KUKA KRL program: MyProgram_229().src

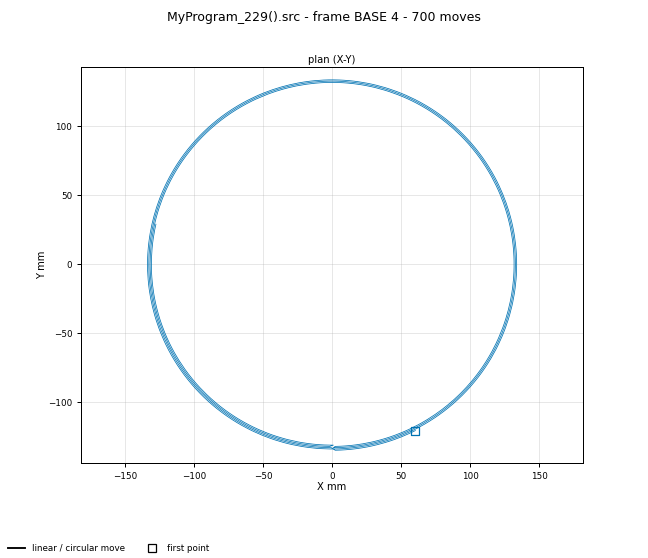
[picture p0: tool path of MyProgram_229().src in frame BASE 4, 700 of 700 moves have a stored position in this frame; points joined in program order, loops and branches not executed]
&ACCESS RVP
&REL 1
&PARAM TEMPLATE = C:\KRC\Roboter\Template\vorgabe
&PARAM EDITMASK = *
DEF MyProgram_229()
; ---- Setting reference (Base) ----
$BASE = BASE_DATA[4]

; --------------------------
; ---- Setting tool (TCP) ----
$TOOL = TOOL_DATA[3]
; --------------------------

$VEL.CP = VEL_APROX_PRINT
Startdeposition()
$VEL.CP = VEL_PRINT
LIN {X 60.3431,Y -120.4102,Z 157,A -66.3783,B 23.115,C -0.9424,E1 23.2036,E2 513.6241} C_DIS
LIN {X 55.6894,Y -122.6317,Z 157,A -68.3242,B 23.1147,C -0.9514,E1 23.1988,E2 515.5416} C_DIS
LIN {X 53.1438,Y -123.7542,Z 157,A -69.519,B 23.1147,C -0.9491,E1 23.1957,E2 516.7391} C_DIS
LIN {X 50.0848,Y -125.0234,Z 157,A -70.9751,B 23.1149,C -0.9447,E1 23.1919,E2 518.2027} C_DIS
LIN {X 44.88,Y -126.987,Z 157,A -73.2835,B 23.1149,C -0.9444,E1 23.1859,E2 520.5065} C_DIS
LIN {X 42.2863,Y -127.8719,Z 157,A -74.8329,B 23.1157,C -0.9239,E1 23.1816,E2 522.1048} C_DIS
LIN {X 38.6503,Y -129.0197,Z 157,A -76.0668,B 23.1151,C -0.9413,E1 23.1785,E2 523.292} C_DIS
LIN {X 32.9154,Y -130.5983,Z 157,A -78.6147,B 23.1151,C -0.9378,E1 23.1716,E2 525.8445} C_DIS
LIN {X 29.0818,Y -131.5067,Z 157,A -80.3833,B 23.1154,C -0.9316,E1 23.1667,E2 527.6262} C_DIS
LIN {X 25.3199,Y -132.2809,Z 157,A -81.9079,B 23.1153,C -0.9357,E1 23.1626,E2 529.1385} C_DIS
LIN {X 21.8715,Y -132.8949,Z 157,A -83.4811,B 23.1155,C -0.9304,E1 23.1582,E2 530.7233} C_DIS
LIN {X 17.6299,Y -133.5236,Z 157,A -85.227,B 23.1154,C -0.933,E1 23.1534,E2 532.4607} C_DIS
LIN {X 14.202,Y -133.9317,Z 157,A -86.7009,B 23.1154,C -0.9319,E1 23.1493,E2 533.9363} C_DIS
LIN {X 10.0398,Y -134.308,Z 157,A -88.4861,B 23.1154,C -0.9307,E1 23.1444,E2 535.7236} C_DIS
LIN {X 6.4164,Y -134.53,Z 157,A -90.0918,B 23.1156,C -0.9271,E1 23.1399,E2 537.3379} C_DIS
LIN {X 2.2217,Y -134.6642,Z 157,A -91.783,B 23.1154,C -0.9312,E1 23.1352,E2 539.0183} C_DIS
LIN {X 2.2217,Y -134.6642,Z 157,A -91.783,B 23.1154,C -0.9312,E1 23.1352,E2 539.0183} C_DIS
Enddeposition()
LIN {X 0.9379,Y -133.7479,Z 157,A -91.7114,B 21.9007,C -0.7569,E1 21.9144,E2 539.2658} C_DIS
Startdeposition()
$VEL.CP = VEL_PRINT
LIN {X 5.092,Y -133.6541,Z 157,A -89.5299,B 21.9,C -0.776,E1 21.9206,E2 537.0334} C_DIS
LIN {X 8.4927,Y -133.4814,Z 157,A -88.065,B 21.9,C -0.7769,E1 21.9247,E2 535.5668} C_DIS
LIN {X 12.2431,Y -133.1905,Z 157,A -86.4619,B 21.9,C -0.7773,E1 21.9292,E2 533.9638} C_DIS
LIN {X 15.7185,Y -132.8241,Z 157,A -84.992,B 21.9,C -0.7769,E1 21.9333,E2 532.4962} C_DIS
LIN {X 18.8317,Y -132.4185,Z 157,A -83.651,B 21.9,C -0.7775,E1 21.937,E2 531.1547} C_DIS
LIN {X 22.9546,Y -131.7678,Z 157,A -81.9321,B 21.9,C -0.7756,E1 21.9417,E2 529.4432} C_DIS
LIN {X 25.8918,Y -131.2232,Z 157,A -80.5104,B 21.8998,C -0.7833,E1 21.9456,E2 528.0027} C_DIS
LIN {X 29.3532,Y -130.4908,Z 157,A -79.0266,B 21.8998,C -0.7832,E1 21.9497,E2 526.5215} C_DIS
LIN {X 32.3293,Y -129.786,Z 157,A -77.8447,B 21.9,C -0.7783,E1 21.9528,E2 525.3545} C_DIS
LIN {X 35.2431,Y -129.0264,Z 157,A -76.4748,B 21.8998,C -0.7834,E1 21.9566,E2 523.9735} C_DIS
LIN {X 38.3629,Y -128.1335,Z 157,A -75.0868,B 21.8998,C -0.7849,E1 21.9603,E2 522.5844} C_DIS
LIN {X 41.4791,Y -127.1589,Z 157,A -73.6902,B 21.8997,C -0.7864,E1 21.964,E2 521.1866} C_DIS
LIN {X 45.073,Y -125.9275,Z 157,A -72.1814,B 21.8998,C -0.7828,E1 21.968,E2 519.691} C_DIS
LIN {X 47.6885,Y -124.9628,Z 157,A -70.8737,B 21.8996,C -0.7898,E1 21.9714,E2 518.3679} C_DIS
LIN {X 51.0833,Y -123.6121,Z 157,A -69.2486,B 21.8994,C -0.7949,E1 21.9756,E2 516.7335} C_DIS
LIN {X 54.2918,Y -122.2364,Z 157,A -68.0057,B 21.8997,C -0.785,E1 21.9787,E2 515.5205} C_DIS
LIN {X 56.898,Y -121.0476,Z 157,A -66.5962,B 21.8994,C -0.7956,E1 21.9824,E2 514.0869} C_DIS
LIN {X 59.9271,Y -119.577,Z 157,A -65.158,B 21.8994,C -0.7977,E1 21.986,E2 512.6475} C_DIS
LIN {X 63.2603,Y -117.8468,Z 157,A -63.4648,B 21.8991,C -0.8045,E1 21.9902,E2 510.9417} C_DIS
LIN {X 66.9687,Y -115.7796,Z 157,A -61.6672,B 21.899,C -0.8067,E1 21.9946,E2 509.1444} C_DIS
LIN {X 70.6246,Y -113.5865,Z 157,A -59.8473,B 21.8989,C -0.8097,E1 21.9989,E2 507.323} C_DIS
LIN {X 74.4235,Y -111.1346,Z 157,A -57.9624,B 21.8989,C -0.811,E1 22.0033,E2 505.442} C_DIS
LIN {X 77.7542,Y -108.8301,Z 157,A -56.1901,B 21.8987,C -0.8163,E1 22.0073,E2 503.6626} C_DIS
LIN {X 81.2948,Y -106.2115,Z 157,A -54.3316,B 21.8986,C -0.8189,E1 22.0115,E2 501.805} C_DIS
LIN {X 84.6122,Y -103.588,Z 157,A -52.512,B 21.8984,C -0.8232,E1 22.0155,E2 499.9819} C_DIS
LIN {X 87.977,Y -100.746,Z 157,A -50.6512,B 21.8983,C -0.8262,E1 22.0194,E2 498.1215} C_DIS
LIN {X 91.1152,Y -97.917,Z 157,A -48.8313,B 21.8981,C -0.8308,E1 22.0232,E2 496.2977} C_DIS
LIN {X 94.3364,Y -94.8176,Z 157,A -46.9545,B 21.8981,C -0.8336,E1 22.0269,E2 494.4228} C_DIS
LIN {X 97.2567,Y -91.8196,Z 157,A -45.1448,B 21.8978,C -0.8388,E1 22.0304,E2 492.6081} C_DIS
LIN {X 100.1751,Y -88.6266,Z 157,A -43.303,B 21.8977,C -0.8429,E1 22.0338,E2 490.7649} C_DIS
LIN {X 103.0497,Y -85.2671,Z 157,A -41.4192,B 21.8975,C -0.8473,E1 22.0372,E2 488.8793} C_DIS
LIN {X 105.6853,Y -81.9776,Z 157,A -39.6275,B 21.8974,C -0.8514,E1 22.0403,E2 487.0864} C_DIS
LIN {X 108.3279,Y -78.4524,Z 157,A -37.7727,B 21.8972,C -0.8549,E1 22.0434,E2 485.2326} C_DIS
LIN {X 110.867,Y -74.8216,Z 157,A -35.9119,B 21.8972,C -0.8583,E1 22.0464,E2 483.3734} C_DIS
LIN {X 113.1329,Y -71.349,Z 157,A -34.1251,B 21.8969,C -0.8638,E1 22.0491,E2 481.5822} C_DIS
LIN {X 115.3011,Y -67.7892,Z 157,A -32.3337,B 21.8967,C -0.8692,E1 22.0516,E2 479.7871} C_DIS
LIN {X 117.4775,Y -63.9435,Z 157,A -30.5231,B 21.8967,C -0.8706,E1 22.0541,E2 477.9836} C_DIS
LIN {X 118.8108,Y -61.4321,Z 157,A -29.1905,B 21.8963,C -0.8799,E1 22.0558,E2 476.6346} C_DIS
LIN {X 120.4363,Y -58.1775,Z 157,A -27.7272,B 21.8963,C -0.8799,E1 22.0576,E2 475.1805} C_DIS
LIN {X 121.9368,Y -54.9615,Z 157,A -26.4378,B 21.8966,C -0.873,E1 22.0591,E2 473.9175} C_DIS
LIN {X 123.0985,Y -52.3132,Z 157,A -25.038,B 21.8961,C -0.8847,E1 22.0606,E2 472.4954} C_DIS
LIN {X 124.3621,Y -49.2338,Z 157,A -23.6241,B 21.896,C -0.8884,E1 22.0621,E2 471.0806} C_DIS
LIN {X 125.5428,Y -46.14,Z 157,A -22.1041,B 21.8956,C -0.8978,E1 22.0636,E2 469.5453} C_DIS
LIN {X 126.7948,Y -42.5725,Z 157,A -20.796,B 21.896,C -0.8874,E1 22.0648,E2 468.2734} C_DIS
LIN {X 127.6564,Y -39.9216,Z 157,A -19.4281,B 21.8955,C -0.8997,E1 22.066,E2 466.8818} C_DIS
LIN {X 128.6609,Y -36.5501,Z 157,A -17.8608,B 21.8952,C -0.9075,E1 22.0672,E2 465.3042} C_DIS
LIN {X 129.5424,Y -33.2894,Z 157,A -16.4631,B 21.8952,C -0.9096,E1 22.0682,E2 463.9101} C_DIS
LIN {X 130.3092,Y -30.1481,Z 157,A -15.1727,B 21.8952,C -0.9093,E1 22.069,E2 462.6291} C_DIS
LIN {X 130.9066,Y -27.4474,Z 157,A -13.9534,B 21.8949,C -0.9147,E1 22.0697,E2 461.4036} C_DIS
LIN {X 131.6022,Y -23.8795,Z 157,A -12.5864,B 21.8951,C -0.9103,E1 22.0704,E2 460.0576} C_DIS
LIN {X 132.0562,Y -21.238,Z 157,A -11.2094,B 21.8945,C -0.9253,E1 22.0711,E2 458.6501} C_DIS
LIN {X 132.5855,Y -17.6196,Z 157,A -9.7043,B 21.8945,C -0.9273,E1 22.0716,E2 457.1499} C_DIS
LIN {X 132.9737,Y -14.3987,Z 157,A -8.3451,B 21.8943,C -0.9303,E1 22.0721,E2 455.7922} C_DIS
LIN {X 133.2838,Y -11.1695,Z 157,A -6.9683,B 21.8942,C -0.9341,E1 22.0724,E2 454.4146} C_DIS
LIN {X 133.5189,Y -7.8835,Z 157,A -5.4562,B 21.8938,C -0.9436,E1 22.0727,E2 452.8876} C_DIS
LIN {X 133.697,Y -3.8022,Z 157,A -3.7923,B 21.8938,C -0.945,E1 22.0729,E2 451.2314} C_DIS
LIN {X 133.7532,Y -0.2268,Z 157,A -2.1342,B 21.8933,C -0.9561,E1 22.0729,E2 449.5551} C_DIS
LIN {X 133.7072,Y 3.4346,Z 157,A -0.713,B 21.8933,C -0.9539,E1 22.0729,E2 448.1497} C_DIS
LIN {X 133.5779,Y 6.8027,Z 157,A 0.707,B 21.8933,C -0.9573,E1 22.0726,E2 446.7303} C_DIS
LIN {X 133.3249,Y 10.683,Z 157,A 2.434,B 21.8929,C -0.9657,E1 22.0723,E2 444.993} C_DIS
LIN {X 132.9986,Y 14.1666,Z 157,A 3.8365,B 21.8929,C -0.9657,E1 22.0719,E2 443.6} C_DIS
LIN {X 132.6097,Y 17.4345,Z 157,A 5.1979,B 21.8928,C -0.9678,E1 22.0714,E2 442.2424} C_DIS
LIN {X 132.1802,Y 20.4373,Z 157,A 6.5397,B 21.8925,C -0.9739,E1 22.0709,E2 440.8933} C_DIS
LIN {X 131.6149,Y 23.8088,Z 157,A 8.0257,B 21.8923,C -0.9796,E1 22.0702,E2 439.4023} C_DIS
LIN {X 130.9066,Y 27.4474,Z 157,A 9.5524,B 21.8923,C -0.9815,E1 22.0693,E2 437.881} C_DIS
LIN {X 130.2144,Y 30.5633,Z 157,A 11.0415,B 21.8918,C -0.9917,E1 22.0684,E2 436.3745} C_DIS
LIN {X 129.301,Y 34.2137,Z 157,A 12.5379,B 21.8918,C -0.991,E1 22.0673,E2 434.8902} C_DIS
LIN {X 128.1335,Y 38.3629,Z 157,A 14.3501,B 21.8916,C -0.9949,E1 22.0659,E2 433.0796} C_DIS
LIN {X 127.0837,Y 41.7048,Z 157,A 15.7518,B 21.8916,C -0.9945,E1 22.0647,E2 431.688} C_DIS
LIN {X 126.1021,Y 44.5887,Z 157,A 17.2854,B 21.891,C -1.0096,E1 22.0633,E2 430.1242} C_DIS
LIN {X 124.7807,Y 48.1571,Z 157,A 18.7673,B 21.891,C -1.0072,E1 22.0619,E2 428.6583} C_DIS
LIN {X 123.607,Y 51.0956,Z 157,A 20.1147,B 21.891,C -1.0107,E1 22.0604,E2 427.3102} C_DIS
LIN {X 122.3341,Y 54.0731,Z 157,A 21.4435,B 21.8909,C -1.0118,E1 22.059,E2 425.9867} C_DIS
LIN {X 121.0476,Y 56.898,Z 157,A 22.8092,B 21.8906,C -1.0173,E1 22.0573,E2 424.615} C_DIS
LIN {X 119.577,Y 59.9271,Z 157,A 24.2433,B 21.8905,C -1.021,E1 22.0556,E2 423.1801} C_DIS
LIN {X 117.8468,Y 63.2603,Z 157,A 25.9173,B 21.8901,C -1.0286,E1 22.0534,E2 421.496} C_DIS
LIN {X 115.7796,Y 66.9687,Z 157,A 27.7258,B 21.8899,C -1.033,E1 22.0509,E2 419.6865} C_DIS
LIN {X 113.5117,Y 70.7447,Z 157,A 29.5907,B 21.8898,C -1.0369,E1 22.0482,E2 417.8221} C_DIS
LIN {X 111.2141,Y 74.3044,Z 157,A 31.3882,B 21.8896,C -1.0408,E1 22.0454,E2 416.0248} C_DIS
LIN {X 108.8301,Y 77.7542,Z 157,A 33.1945,B 21.8894,C -1.0458,E1 22.0425,E2 414.2154} C_DIS
LIN {X 106.1216,Y 81.4123,Z 157,A 35.0886,B 21.8893,C -1.0479,E1 22.0393,E2 412.3262} C_DIS
LIN {X 103.5981,Y 84.6,Z 157,A 36.8664,B 21.889,C -1.0538,E1 22.0362,E2 410.5422} C_DIS
LIN {X 100.7114,Y 88.0167,Z 157,A 38.7432,B 21.8889,C -1.0563,E1 22.0328,E2 408.6685} C_DIS
LIN {X 97.917,Y 91.1152,Z 157,A 40.5506,B 21.8887,C -1.0613,E1 22.0294,E2 406.857} C_DIS
LIN {X 94.7695,Y 94.3847,Z 157,A 42.4807,B 21.8885,C -1.0649,E1 22.0256,E2 404.9269} C_DIS
LIN {X 91.8196,Y 97.2567,Z 157,A 44.2396,B 21.8883,C -1.0683,E1 22.0221,E2 403.1672} C_DIS
LIN {X 88.5047,Y 100.2829,Z 157,A 46.1587,B 21.8882,C -1.072,E1 22.0181,E2 401.2472} C_DIS
LIN {X 85.2671,Y 103.0497,Z 157,A 47.9486,B 21.8881,C -1.0739,E1 22.0143,E2 399.4603} C_DIS
LIN {X 81.9776,Y 105.6853,Z 157,A 49.7695,B 21.8879,C -1.078,E1 22.0103,E2 397.6363} C_DIS
LIN {X 78.312,Y 108.4297,Z 157,A 51.6684,B 21.8879,C -1.0785,E1 22.006,E2 395.744} C_DIS
LIN {X 74.97,Y 110.7665,Z 157,A 53.4546,B 21.8876,C -1.0833,E1 22.0019,E2 393.9521} C_DIS
LIN {X 71.349,Y 113.1329,Z 157,A 55.2818,B 21.8876,C -1.085,E1 21.9976,E2 392.1272} C_DIS
LIN {X 67.7892,Y 115.3011,Z 157,A 57.079,B 21.8874,C -1.0882,E1 21.9933,E2 390.3278} C_DIS
LIN {X 63.873,Y 117.516,Z 157,A 58.9688,B 21.8874,C -1.0891,E1 21.9887,E2 388.4419} C_DIS
LIN {X 59.9271,Y 119.577,Z 157,A 60.8232,B 21.8874,C -1.0891,E1 21.9841,E2 386.5933} C_DIS
LIN {X 56.5595,Y 121.2041,Z 157,A 62.3941,B 21.8874,C -1.0897,E1 21.9801,E2 385.0258} C_DIS
LIN {X 53.8464,Y 122.4356,Z 157,A 63.6907,B 21.8872,C -1.0921,E1 21.9768,E2 383.7265} C_DIS
LIN {X 50.7755,Y 123.7406,Z 157,A 65.2625,B 21.8868,C -1.1003,E1 21.9727,E2 382.137} C_DIS
LIN {X 47.2895,Y 125.1123,Z 157,A 66.7188,B 21.8871,C -1.095,E1 21.969,E2 380.6986} C_DIS
LIN {X 44.1628,Y 126.2498,Z 157,A 67.963,B 21.8874,C -1.0879,E1 21.9658,E2 379.4765} C_DIS
LIN {X 41.4791,Y 127.1589,Z 157,A 69.4179,B 21.8868,C -1.1001,E1 21.9618,E2 377.9921} C_DIS
LIN {X 38.2927,Y 128.154,Z 157,A 70.742,B 21.887,C -1.0963,E1 21.9583,E2 376.6809} C_DIS
LIN {X 34.7348,Y 129.162,Z 157,A 72.34,B 21.887,C -1.098,E1 21.954,E2 375.0812} C_DIS
LIN {X 32.1228,Y 129.8385,Z 157,A 73.5018,B 21.8869,C -1.099,E1 21.9509,E2 373.9189} C_DIS
LIN {X 29.0047,Y 130.5704,Z 157,A 74.8696,B 21.8869,C -1.0996,E1 21.9471,E2 372.5518} C_DIS
LIN {X 25.6745,Y 131.2647,Z 157,A 76.4136,B 21.8866,C -1.1043,E1 21.9429,E2 370.9973} C_DIS
LIN {X 22.1019,Y 131.9121,Z 157,A 77.8735,B 21.8868,C -1.1005,E1 21.9389,E2 369.5493} C_DIS
LIN {X 18.9582,Y 132.4005,Z 157,A 79.2567,B 21.8868,C -1.1018,E1 21.9351,E2 368.164} C_DIS
LIN {X 15.7544,Y 132.8198,Z 157,A 80.6144,B 21.8868,C -1.101,E1 21.9313,E2 366.8099} C_DIS
LIN {X 12.3778,Y 133.1776,Z 157,A 82.1416,B 21.8866,C -1.1045,E1 21.9271,E2 365.2743} C_DIS
LIN {X 8.6379,Y 133.4724,Z 157,A 83.7484,B 21.8866,C -1.1045,E1 21.9226,E2 363.6682} C_DIS
LIN {X 5.0791,Y 133.6546,Z 157,A 85.2614,B 21.8866,C -1.1039,E1 21.9184,E2 362.1575} C_DIS
LIN {X 1.1299,Y 133.7469,Z 157,A 86.9566,B 21.8866,C -1.1039,E1 21.9136,E2 360.4627} C_DIS
LIN {X -2.4434,Y 133.7289,Z 157,A 88.5191,B 21.8866,C -1.105,E1 21.9093,E2 358.8971} C_DIS
LIN {X -6.2756,Y 133.6044,Z 157,A 90.1048,B 21.8867,C -1.1019,E1 21.9049,E2 357.3192} C_DIS
LIN {X -9.6506,Y 133.4024,Z 157,A 91.5167,B 21.8869,C -1.0998,E1 21.9009,E2 355.9127} C_DIS
LIN {X -12.8698,Y 133.1303,Z 157,A 92.905,B 21.8869,C -1.0993,E1 21.8971,E2 354.5247} C_DIS
LIN {X -16.0354,Y 132.7863,Z 157,A 94.3332,B 21.8868,C -1.1015,E1 21.8931,E2 353.0896} C_DIS
LIN {X -20.2505,Y 132.2091,Z 157,A 96.0945,B 21.887,C -1.0976,E1 21.8883,E2 351.3371} C_DIS
LIN {X -24.3381,Y 131.5202,Z 157,A 98.0394,B 21.8867,C -1.1039,E1 21.8829,E2 349.3731} C_DIS
LIN {X -27.4474,Y 130.9066,Z 157,A 99.2452,B 21.887,C -1.096,E1 21.8796,E2 348.1869} C_DIS
LIN {X -30.5633,Y 130.2144,Z 157,A 100.7348,B 21.8868,C -1.1002,E1 21.8755,E2 346.6836} C_DIS
LIN {X -34.2322,Y 129.296,Z 157,A 102.0255,B 21.8876,C -1.0841,E1 21.8721,E2 345.4342} C_DIS
LIN {X -36.8033,Y 128.5901,Z 157,A 103.3903,B 21.8872,C -1.0927,E1 21.8684,E2 344.0436} C_DIS
LIN {X -39.9216,Y 127.6564,Z 157,A 104.7903,B 21.8872,C -1.0915,E1 21.8647,E2 342.6442} C_DIS
LIN {X -43.0349,Y 126.6408,Z 157,A 106.199,B 21.8873,C -1.0901,E1 21.8609,E2 341.2362} C_DIS
LIN {X -46.2916,Y 125.486,Z 157,A 107.7634,B 21.8873,C -1.092,E1 21.8568,E2 339.6631} C_DIS
LIN {X -49.2338,Y 124.3621,Z 157,A 109.0406,B 21.8875,C -1.087,E1 21.8535,E2 338.3961} C_DIS
LIN {X -52.3132,Y 123.0985,Z 157,A 110.575,B 21.8873,C -1.0898,E1 21.8495,E2 336.8501} C_DIS
LIN {X -55.7045,Y 121.5995,Z 157,A 112.1216,B 21.8875,C -1.0857,E1 21.8456,E2 335.3102} C_DIS
LIN {X -58.7926,Y 120.1366,Z 157,A 113.3776,B 21.8881,C -1.0743,E1 21.8425,E2 334.0811} C_DIS
LIN {X -61.4321,Y 118.8108,Z 157,A 114.8984,B 21.8876,C -1.0834,E1 21.8387,E2 332.5309} C_DIS
LIN {X -65.1638,Y 116.8058,Z 157,A 116.7225,B 21.8878,C -1.0808,E1 21.8342,E2 330.708} C_DIS
LIN {X -68.8461,Y 114.6739,Z 157,A 118.5547,B 21.8878,C -1.078,E1 21.8298,E2 328.8769} C_DIS
LIN {X -72.4729,Y 112.417,Z 157,A 120.4124,B 21.888,C -1.0758,E1 21.8254,E2 327.0182} C_DIS
LIN {X -76.0378,Y 110.0371,Z 157,A 122.2726,B 21.8881,C -1.0733,E1 21.8211,E2 325.1575} C_DIS
LIN {X -79.5346,Y 107.5368,Z 157,A 124.11,B 21.8883,C -1.0694,E1 21.817,E2 323.3232} C_DIS
LIN {X -82.9573,Y 104.9189,Z 157,A 125.9478,B 21.8885,C -1.0651,E1 21.8129,E2 321.489} C_DIS
LIN {X -86.3311,Y 102.1607,Z 157,A 127.833,B 21.8886,C -1.0619,E1 21.8089,E2 319.6042} C_DIS
LIN {X -89.5574,Y 99.3447,Z 157,A 129.6699,B 21.8888,C -1.0578,E1 21.8051,E2 317.7698} C_DIS
LIN {X -92.7237,Y 96.3961,Z 157,A 131.5524,B 21.889,C -1.0548,E1 21.8012,E2 315.8866} C_DIS
LIN {X -95.8566,Y 93.281,Z 157,A 133.4143,B 21.8892,C -1.0489,E1 21.7976,E2 314.0312} C_DIS
LIN {X -98.7633,Y 90.1981,Z 157,A 135.263,B 21.8894,C -1.0459,E1 21.7941,E2 312.1812} C_DIS
LIN {X -101.6273,Y 86.9586,Z 157,A 137.1446,B 21.8895,C -1.0425,E1 21.7906,E2 310.299} C_DIS
LIN {X -104.4239,Y 83.5793,Z 157,A 138.9987,B 21.8898,C -1.0365,E1 21.7874,E2 308.451} C_DIS
LIN {X -107.0225,Y 80.2252,Z 157,A 140.8629,B 21.8899,C -1.0337,E1 21.7842,E2 306.584} C_DIS
LIN {X -109.5466,Y 76.7428,Z 157,A 142.7108,B 21.8901,C -1.0289,E1 21.7812,E2 304.7385} C_DIS
LIN {X -111.9804,Y 73.1453,Z 157,A 144.5738,B 21.8904,C -1.0239,E1 21.7784,E2 302.8783} C_DIS
LIN {X -114.2325,Y 69.5761,Z 157,A 146.4327,B 21.8904,C -1.021,E1 21.7756,E2 301.0162} C_DIS
LIN {X -116.4578,Y 65.7828,Z 157,A 148.2479,B 21.8909,C -1.0127,E1 21.7731,E2 299.2124} C_DIS
LIN {X -118.0241,Y 62.9303,Z 157,A 149.5975,B 21.8911,C -1.0067,E1 21.7713,E2 297.8706} C_DIS
LIN {X -119.577,Y 59.9271,Z 157,A 151.0547,B 21.8913,C -1.0029,E1 21.7695,E2 296.4148} C_DIS
LIN {X -121.0476,Y 56.898,Z 157,A 152.6587,B 21.8912,C -1.0055,E1 21.7676,E2 294.7938} C_DIS
LIN {X -122.4356,Y 53.8464,Z 157,A 153.951,B 21.8916,C -0.995,E1 21.7661,E2 293.5213} C_DIS
LIN {X -123.7406,Y 50.7755,Z 157,A 155.3893,B 21.8918,C -0.9911,E1 21.7646,E2 292.0844} C_DIS
LIN {X -124.9628,Y 47.6885,Z 157,A 156.8917,B 21.8918,C -0.9901,E1 21.763,E2 290.5747} C_DIS
LIN {X -126.1782,Y 44.3693,Z 157,A 158.2547,B 21.8923,C -0.9791,E1 21.7618,E2 289.2326} C_DIS
LIN {X -127.1589,Y 41.4791,Z 157,A 159.6595,B 21.8923,C -0.9791,E1 21.7605,E2 287.8184} C_DIS
LIN {X -128.1335,Y 38.3629,Z 157,A 161.0668,B 21.8925,C -0.9752,E1 21.7594,E2 286.4124} C_DIS
LIN {X -129.0264,Y 35.2431,Z 157,A 162.6053,B 21.8924,C -0.9771,E1 21.7582,E2 284.8583} C_DIS
LIN {X -129.8852,Y 31.929,Z 157,A 163.8646,B 21.893,C -0.9637,E1 21.7574,E2 283.6266} C_DIS
LIN {X -130.5704,Y 29.0047,Z 157,A 165.2353,B 21.893,C -0.9632,E1 21.7565,E2 282.248} C_DIS
LIN {X -131.2478,Y 25.763,Z 157,A 166.6121,B 21.8932,C -0.9569,E1 21.7558,E2 280.8787} C_DIS
LIN {X -131.7978,Y 22.7868,Z 157,A 167.9668,B 21.8933,C -0.9552,E1 21.7551,E2 279.5192} C_DIS
LIN {X -132.3784,Y 19.1128,Z 157,A 169.5584,B 21.8935,C -0.9501,E1 21.7544,E2 277.9305} C_DIS
LIN {X -132.9008,Y 15.0757,Z 157,A 171.3238,B 21.8937,C -0.9454,E1 21.7538,E2 276.1655} C_DIS
LIN {X -133.2121,Y 12.0183,Z 157,A 172.6483,B 21.8939,C -0.9415,E1 21.7535,E2 274.8423} C_DIS
LIN {X -133.4804,Y 8.5087,Z 157,A 174.2102,B 21.8939,C -0.939,E1 21.7532,E2 273.2763} C_DIS
LIN {X -133.6528,Y 5.126,Z 157,A 175.6847,B 21.8941,C -0.9354,E1 21.753,E2 271.8014} C_DIS
LIN {X -133.7449,Y 1.4811,Z 157,A 177.2307,B 21.8944,C -0.9296,E1 21.753,E2 270.2599} C_DIS
LIN {X -133.7449,Y -1.4811,Z 157,A 178.4753,B 21.8946,C -0.9245,E1 21.753,E2 269.0204} C_DIS
LIN {X -133.668,Y -4.7371,Z 157,A 179.9599,B 21.8946,C -0.9239,E1 21.753,E2 267.5272} C_DIS
LIN {X -133.4999,Y -8.1911,Z 157,A -178.6104,B 21.8949,C -0.917,E1 21.7533,E2 266.1062} C_DIS
LIN {X -133.2838,Y -11.1695,Z 157,A -177.2945,B 21.8949,C -0.9145,E1 21.7536,E2 264.7879} C_DIS
LIN {X -132.953,Y -14.5903,Z 157,A -175.7971,B 21.8951,C -0.9109,E1 21.754,E2 263.2897} C_DIS
LIN {X -132.516,Y -18.1497,Z 157,A -174.1411,B 21.8951,C -0.9111,E1 21.7546,E2 261.6217} C_DIS
LIN {X -131.9747,Y -21.7267,Z 157,A -172.9189,B 21.8958,C -0.8924,E1 21.7551,E2 260.4416} C_DIS
LIN {X -131.5202,Y -24.3381,Z 157,A -171.582,B 21.8956,C -0.8973,E1 21.7558,E2 259.0821} C_DIS
LIN {X -130.9014,Y -27.4717,Z 157,A -170.211,B 21.8958,C -0.8932,E1 21.7565,E2 257.7128} C_DIS
LIN {X -130.2144,Y -30.5633,Z 157,A -168.6872,B 21.8957,C -0.8962,E1 21.7575,E2 256.1707} C_DIS
LIN {X -129.3021,Y -34.2095,Z 157,A -167.4184,B 21.8964,C -0.8767,E1 21.7584,E2 254.9458} C_DIS
LIN {X -128.5901,Y -36.8033,Z 157,A -166.046,B 21.8962,C -0.8826,E1 21.7594,E2 253.5484} C_DIS
LIN {X -127.4949,Y -40.4272,Z 157,A -164.3885,B 21.8963,C -0.8793,E1 21.7608,E2 251.8887} C_DIS
LIN {X -126.4671,Y -43.5359,Z 157,A -163.1999,B 21.8968,C -0.8659,E1 21.7618,E2 250.7282} C_DIS
LIN {X -125.5428,Y -46.14,Z 157,A -161.8021,B 21.8966,C -0.8716,E1 21.7632,E2 249.306} C_DIS
LIN {X -124.2433,Y -49.5285,Z 157,A -160.1997,B 21.8967,C -0.8691,E1 21.7648,E2 247.6999} C_DIS
LIN {X -122.8926,Y -52.7892,Z 157,A -158.9102,B 21.8972,C -0.8552,E1 21.7662,E2 246.4396} C_DIS
LIN {X -121.7519,Y -55.3748,Z 157,A -157.4906,B 21.897,C -0.8607,E1 21.7678,E2 244.9961} C_DIS
LIN {X -120.3226,Y -58.4156,Z 157,A -156.0401,B 21.8972,C -0.8571,E1 21.7695,E2 243.546} C_DIS
LIN {X -118.5872,Y -61.8579,Z 157,A -154.3605,B 21.8972,C -0.8538,E1 21.7717,E2 241.865} C_DIS
LIN {X -116.5735,Y -65.5769,Z 157,A -152.4954,B 21.8974,C -0.8512,E1 21.7742,E2 239.9957} C_DIS
LIN {X -114.4255,Y -69.2569,Z 157,A -150.6576,B 21.8975,C -0.8469,E1 21.7768,E2 238.1585} C_DIS
LIN {X -112.0931,Y -72.9719,Z 157,A -148.7857,B 21.8977,C -0.8417,E1 21.7796,E2 236.2896} C_DIS
LIN {X -109.8202,Y -76.3495,Z 157,A -146.9891,B 21.8978,C -0.8396,E1 21.7825,E2 234.4884} C_DIS
LIN {X -107.1666,Y -80.0316,Z 157,A -145.0767,B 21.898,C -0.8334,E1 21.7856,E2 232.582} C_DIS
LIN {X -104.6813,Y -83.2558,Z 157,A -143.2775,B 21.8981,C -0.8316,E1 21.7887,E2 230.7777} C_DIS
LIN {X -101.8748,Y -86.6675,Z 157,A -141.3937,B 21.8983,C -0.8268,E1 21.7921,E2 228.8967} C_DIS
LIN {X -99.0204,Y -89.9148,Z 157,A -139.5312,B 21.8984,C -0.8231,E1 21.7956,E2 227.0346} C_DIS
LIN {X -95.9992,Y -93.1337,Z 157,A -137.646,B 21.8986,C -0.8187,E1 21.7992,E2 225.1518} C_DIS
LIN {X -92.9987,Y -96.1299,Z 157,A -135.8043,B 21.8986,C -0.816,E1 21.8029,E2 223.3084} C_DIS
LIN {X -89.745,Y -99.1745,Z 157,A -133.9094,B 21.8988,C -0.8115,E1 21.8067,E2 221.4167} C_DIS
LIN {X -86.6675,Y -101.8748,Z 157,A -132.1048,B 21.8988,C -0.8103,E1 21.8106,E2 219.6071} C_DIS
LIN {X -83.22,Y -104.7099,Z 157,A -130.2056,B 21.899,C -0.8062,E1 21.8147,E2 217.7107} C_DIS
LIN {X -79.8004,Y -107.3388,Z 157,A -128.3591,B 21.8991,C -0.8028,E1 21.8188,E2 215.8655} C_DIS
LIN {X -76.3495,Y -109.8202,Z 157,A -126.5058,B 21.8991,C -0.8012,E1 21.823,E2 214.0092} C_DIS
LIN {X -72.5888,Y -112.3418,Z 157,A -124.6167,B 21.8994,C -0.7959,E1 21.8274,E2 212.1274} C_DIS
LIN {X -69.1689,Y -114.4787,Z 157,A -122.8446,B 21.8994,C -0.7953,E1 21.8316,E2 210.3505} C_DIS
LIN {X -65.3527,Y -116.6996,Z 157,A -120.9761,B 21.8995,C -0.7916,E1 21.8362,E2 208.4855} C_DIS
LIN {X -62.0945,Y -118.4629,Z 157,A -119.4964,B 21.8997,C -0.7847,E1 21.8398,E2 207.0196} C_DIS
LIN {X -59.5103,Y -119.7825,Z 157,A -118.2053,B 21.8997,C -0.7853,E1 21.843,E2 205.7229} C_DIS
LIN {X -56.8387,Y -121.075,Z 157,A -116.9185,B 21.8997,C -0.7844,E1 21.8463,E2 204.4346} C_DIS
LIN {X -53.4278,Y -122.6166,Z 157,A -115.3225,B 21.8998,C -0.7823,E1 21.8503,E2 202.8398} C_DIS
LIN {X -50.7755,Y -123.7406,Z 157,A -114.0518,B 21.8998,C -0.7826,E1 21.8536,E2 201.5648} C_DIS
LIN {X -47.3519,Y -125.0889,Z 157,A -112.6109,B 21.9001,C -0.775,E1 21.8573,E2 200.1409} C_DIS
LIN {X -44.5887,Y -126.1021,Z 157,A -111.1089,B 21.8997,C -0.7848,E1 21.8613,E2 198.6091} C_DIS
LIN {X -41.4742,Y -127.1605,Z 157,A -109.8036,B 21.8999,C -0.7789,E1 21.8648,E2 197.3168} C_DIS
LIN {X -37.9147,Y -128.2647,Z 157,A -108.2065,B 21.8999,C -0.7778,E1 21.869,E2 195.7195} C_DIS
LIN {X -35.2431,Y -129.0264,Z 157,A -107.014,B 21.9,C -0.7771,E1 21.8723,E2 194.5268} C_DIS
LIN {X -32.1228,Y -129.8385,Z 157,A -105.6328,B 21.9,C -0.7763,E1 21.876,E2 193.1455} C_DIS
LIN {X -28.6659,Y -130.6435,Z 157,A -104.0411,B 21.9,C -0.7788,E1 21.8803,E2 191.5447} C_DIS
LIN {X -25.2034,Y -131.3548,Z 157,A -102.5851,B 21.9,C -0.7755,E1 21.8843,E2 190.0956} C_DIS
LIN {X -22.0716,Y -131.9171,Z 157,A -101.2437,B 21.9001,C -0.774,E1 21.888,E2 188.7567} C_DIS
LIN {X -17.6282,Y -132.5843,Z 157,A -99.2771,B 21.9001,C -0.7755,E1 21.8935,E2 186.7843} C_DIS
LIN {X -14.3698,Y -132.9768,Z 157,A -97.9181,B 21.9001,C -0.7731,E1 21.8972,E2 185.4307} C_DIS
LIN {X -11.1695,Y -133.2838,Z 157,A -96.5368,B 21.9001,C -0.7731,E1 21.9011,E2 184.0484} C_DIS
LIN {X -8.3117,Y -133.4925,Z 157,A -95.2657,B 21.9001,C -0.7752,E1 21.9046,E2 182.7714} C_DIS
LIN {X -4.4627,Y -133.6787,Z 157,A -93.5354,B 21.8999,C -0.779,E1 21.9095,E2 181.0306} C_DIS
LIN {X -1.4811,Y -133.7449,Z 157,A -92.3889,B 21.9001,C -0.7731,E1 21.9126,E2 179.8998} C_DIS
LIN {X 0.9379,Y -133.7479,Z 157,A -91.7109,B 21.9007,C -0.7567,E1 21.9144,E2 179.2658} C_DIS
Enddeposition()
LIN {X 0.9379,Y -133.7479,Z 157,A -91.7109,B 21.9007,C -0.7567,E1 21.9144,E2 179.2658} C_DIS
Startdeposition()
$VEL.CP = VEL_PRINT
LIN {X -0.5639,Y -132.8185,Z 157,A -92.3139,B 20.8222,C -0.5947,E1 20.829,E2 180.2014} C_DIS
LIN {X -4.6102,Y -132.7407,Z 157,A -94.1013,B 20.8222,C -0.5927,E1 20.824,E2 181.9946} C_DIS
LIN {X -8.567,Y -132.5435,Z 157,A -95.8253,B 20.8222,C -0.592,E1 20.8192,E2 183.7211} C_DIS
LIN {X -12.7955,Y -132.2017,Z 157,A -97.5963,B 20.8222,C -0.5947,E1 20.8142,E2 185.4855} C_DIS
LIN {X -16.9939,Y -131.728,Z 157,A -99.3619,B 20.8222,C -0.5975,E1 20.8094,E2 187.2447} C_DIS
LIN {X -21.0982,Y -131.1352,Z 157,A -101.3069,B 20.8223,C -0.5913,E1 20.8039,E2 189.2093} C_DIS
LIN {X -24.7514,Y -130.4928,Z 157,A -102.8249,B 20.8222,C -0.5954,E1 20.7998,E2 190.7175} C_DIS
LIN {X -28.4496,Y -129.7373,Z 157,A -104.4155,B 20.8222,C -0.5978,E1 20.7955,E2 192.3039} C_DIS
LIN {X -32.299,Y -128.8327,Z 157,A -106.033,B 20.822,C -0.6025,E1 20.7911,E2 193.9109} C_DIS
LIN {X -36.5783,Y -127.6854,Z 157,A -108.1843,B 20.8222,C -0.5935,E1 20.7852,E2 196.0914} C_DIS
LIN {X -41.6451,Y -126.1218,Z 157,A -110.3657,B 20.8221,C -0.5998,E1 20.7795,E2 198.26} C_DIS
LIN {X -44.9014,Y -124.9992,Z 157,A -111.7913,B 20.822,C -0.6036,E1 20.7757,E2 199.6781} C_DIS
LIN {X -47.9748,Y -123.8521,Z 157,A -113.2835,B 20.822,C -0.6017,E1 20.7718,E2 201.1796} C_DIS
LIN {X -52.1777,Y -122.1422,Z 157,A -115.2841,B 20.822,C -0.6019,E1 20.7666,E2 203.1851} C_DIS
LIN {X -55.0391,Y -120.8809,Z 157,A -116.6652,B 20.822,C -0.6021,E1 20.7631,E2 204.5699} C_DIS
LIN {X -58.3945,Y -119.2943,Z 157,A -118.1358,B 20.8218,C -0.6095,E1 20.7594,E2 206.0243} C_DIS
LIN {X -61.3221,Y -117.8164,Z 157,A -119.6292,B 20.8218,C -0.608,E1 20.7557,E2 207.5268} C_DIS
LIN {X -65.3063,Y -115.6571,Z 157,A -121.6101,B 20.8218,C -0.6095,E1 20.7509,E2 209.5102} C_DIS
LIN {X -69.1678,Y -113.3902,Z 157,A -123.6026,B 20.8218,C -0.6098,E1 20.7461,E2 211.5094} C_DIS
LIN {X -72.9063,Y -111.023,Z 157,A -125.4971,B 20.8217,C -0.6134,E1 20.7416,E2 213.4012} C_DIS
LIN {X -76.6922,Y -108.4423,Z 157,A -127.4739,B 20.8217,C -0.6167,E1 20.7371,E2 215.3771} C_DIS
LIN {X -80.3004,Y -105.7988,Z 157,A -129.4221,B 20.8215,C -0.6192,E1 20.7327,E2 217.3265} C_DIS
LIN {X -83.6759,Y -103.1498,Z 157,A -131.2622,B 20.8215,C -0.6231,E1 20.7287,E2 219.1642} C_DIS
LIN {X -86.9067,Y -100.4426,Z 157,A -133.1161,B 20.8214,C -0.6251,E1 20.7248,E2 221.0212} C_DIS
LIN {X -89.7534,Y -97.9069,Z 157,A -134.612,B 20.8211,C -0.6344,E1 20.7217,E2 222.498} C_DIS
LIN {X -95.1558,Y -92.6657,Z 157,A -138.0588,B 20.8211,C -0.633,E1 20.7148,E2 225.9665} C_DIS
LIN {X -98.1987,Y -89.4342,Z 157,A -139.9325,B 20.821,C -0.6389,E1 20.7113,E2 227.8337} C_DIS
LIN {X -101.0482,Y -86.2016,Z 157,A -141.6695,B 20.8207,C -0.6481,E1 20.7081,E2 229.5545} C_DIS
LIN {X -103.5211,Y -83.2156,Z 157,A -143.4668,B 20.8207,C -0.6469,E1 20.7049,E2 231.3652} C_DIS
LIN {X -106.2221,Y -79.7394,Z 157,A -145.4216,B 20.8207,C -0.6493,E1 20.7016,E2 233.3248} C_DIS
LIN {X -108.8015,Y -76.1826,Z 157,A -147.3539,B 20.8206,C -0.6525,E1 20.6985,E2 235.2596} C_DIS
LIN {X -110.4733,Y -73.7364,Z 157,A -148.7381,B 20.8206,C -0.6514,E1 20.6963,E2 236.6552} C_DIS
LIN {X -113.2608,Y -69.3787,Z 157,A -150.8197,B 20.8202,C -0.6632,E1 20.6932,E2 238.7165} C_DIS
LIN {X -115.4163,Y -65.7305,Z 157,A -152.719,B 20.8202,C -0.6652,E1 20.6906,E2 240.6222} C_DIS
LIN {X -117.4116,Y -62.0931,Z 157,A -154.3932,B 20.8199,C -0.6747,E1 20.6884,E2 242.2806} C_DIS
LIN {X -118.8072,Y -59.382,Z 157,A -155.7944,B 20.8199,C -0.6748,E1 20.6866,E2 243.6904} C_DIS
LIN {X -121.3389,Y -54.0167,Z 157,A -158.3429,B 20.8196,C -0.6825,E1 20.6836,E2 246.2345} C_DIS
LIN {X -123.0663,Y -49.9568,Z 157,A -160.2462,B 20.8195,C -0.6879,E1 20.6815,E2 248.1353} C_DIS
LIN {X -124.1172,Y -47.2904,Z 157,A -161.8269,B 20.8198,C -0.6778,E1 20.6799,E2 249.7554} C_DIS
LIN {X -125.3266,Y -43.9819,Z 157,A -163.0141,B 20.8192,C -0.6954,E1 20.6789,E2 250.9011} C_DIS
LIN {X -126.4866,Y -40.5224,Z 157,A -164.5693,B 20.8191,C -0.7008,E1 20.6775,E2 252.4519} C_DIS
LIN {X -127.427,Y -37.4607,Z 157,A -165.9742,B 20.819,C -0.704,E1 20.6764,E2 253.8577} C_DIS
LIN {X -128.3403,Y -34.2008,Z 157,A -167.43,B 20.8188,C -0.7086,E1 20.6753,E2 255.3109} C_DIS
LIN {X -129.1063,Y -31.1851,Z 157,A -168.8148,B 20.8188,C -0.711,E1 20.6744,E2 256.6989} C_DIS
LIN {X -129.7675,Y -28.3096,Z 157,A -171.1157,B 20.8199,C -0.6748,E1 20.673,E2 259.1189} C_DIS
LIN {X -131.0953,Y -21.3375,Z 157,A -173.0817,B 20.8182,C -0.7269,E1 20.6721,E2 260.9517} C_DIS
LIN {X -132.0191,Y -14.5629,Z 157,A -176.1597,B 20.8181,C -0.731,E1 20.671,E2 264.0405} C_DIS
LIN {X -132.5292,Y -8.7988,Z 157,A -178.7361,B 20.8179,C -0.7357,E1 20.6704,E2 266.6226} C_DIS
LIN {X -132.7204,Y -5.1317,Z 157,A 179.7205,B 20.8177,C -0.7423,E1 20.6702,E2 268.1587} C_DIS
LIN {X -132.8172,Y -0.9149,Z 157,A 177.9018,B 20.8175,C -0.7481,E1 20.6702,E2 269.9744} C_DIS
LIN {X -132.7867,Y 3.0201,Z 157,A 176.1217,B 20.8175,C -0.7502,E1 20.6702,E2 271.7617} C_DIS
LIN {X -132.644,Y 6.8277,Z 157,A 174.5144,B 20.8172,C -0.7569,E1 20.6704,E2 273.3619} C_DIS
LIN {X -132.3603,Y 11.0349,Z 157,A 172.7374,B 20.8169,C -0.7643,E1 20.6708,E2 275.131} C_DIS
LIN {X -132.1039,Y 13.7754,Z 157,A 171.6388,B 20.8167,C -0.7715,E1 20.6711,E2 276.2172} C_DIS
LIN {X -131.4133,Y 19.2812,Z 157,A 168.2077,B 20.8178,C -0.7388,E1 20.6724,E2 279.7663} C_DIS
LIN {X -130.3407,Y 25.5471,Z 157,A 166.3577,B 20.8163,C -0.782,E1 20.6733,E2 281.5072} C_DIS
LIN {X -129.2266,Y 30.686,Z 157,A 164.0286,B 20.8161,C -0.7867,E1 20.6747,E2 283.8397} C_DIS
LIN {X -128.3836,Y 34.0388,Z 157,A 162.5579,B 20.8159,C -0.7922,E1 20.6758,E2 285.3055} C_DIS
LIN {X -127.4901,Y 37.2454,Z 157,A 161.0713,B 20.8159,C -0.7947,E1 20.6769,E2 286.7957} C_DIS
LIN {X -126.3709,Y 40.8848,Z 157,A 159.3655,B 20.8157,C -0.7972,E1 20.6783,E2 288.5063} C_DIS
LIN {X -125.0163,Y 44.854,Z 157,A 157.6297,B 20.8154,C -0.8056,E1 20.6799,E2 290.2303} C_DIS
LIN {X -123.7374,Y 48.27,Z 157,A 156.037,B 20.8153,C -0.8096,E1 20.6815,E2 291.8228} C_DIS
LIN {X -122.2101,Y 52.0207,Z 157,A 154.1633,B 20.8153,C -0.8098,E1 20.6835,E2 293.7085} C_DIS
LIN {X -121.0792,Y 54.5974,Z 157,A 152.9868,B 20.8151,C -0.8149,E1 20.6849,E2 294.8786} C_DIS
LIN {X -118.6652,Y 59.6649,Z 157,A 150.3028,B 20.8152,C -0.8117,E1 20.6882,E2 297.5895} C_DIS
LIN {X -117.1077,Y 62.6677,Z 157,A 148.9573,B 20.8149,C -0.8203,E1 20.6899,E2 298.9193} C_DIS
LIN {X -114.7091,Y 66.9578,Z 157,A 146.893,B 20.8146,C -0.8285,E1 20.6928,E2 300.9737} C_DIS
LIN {X -112.4101,Y 70.7489,Z 157,A 145.0008,B 20.8143,C -0.8346,E1 20.6955,E2 302.8604} C_DIS
LIN {X -110.0113,Y 74.4239,Z 157,A 143.0922,B 20.8142,C -0.8392,E1 20.6985,E2 304.7678} C_DIS
LIN {X -107.3677,Y 78.19,Z 157,A 141.0731,B 20.814,C -0.8432,E1 20.7018,E2 306.7878} C_DIS
LIN {X -104.7191,Y 81.7037,Z 157,A 139.139,B 20.8139,C -0.8467,E1 20.7051,E2 308.7232} C_DIS
LIN {X -101.8852,Y 85.2107,Z 157,A 137.2269,B 20.8136,C -0.853,E1 20.7084,E2 310.6284} C_DIS
LIN {X -99.1034,Y 88.4306,Z 157,A 135.3876,B 20.8135,C -0.8574,E1 20.7118,E2 312.4653} C_DIS
LIN {X -96.1611,Y 91.6214,Z 157,A 133.4723,B 20.8133,C -0.8602,E1 20.7155,E2 314.3829} C_DIS
LIN {X -92.8711,Y 94.9547,Z 157,A 131.4624,B 20.8131,C -0.8654,E1 20.7194,E2 316.3886} C_DIS
LIN {X -89.7787,Y 97.8836,Z 157,A 129.6612,B 20.8129,C -0.871,E1 20.7231,E2 318.1829} C_DIS
LIN {X -86.578,Y 100.7258,Z 157,A 127.7599,B 20.8129,C -0.8729,E1 20.7271,E2 320.0881} C_DIS
LIN {X -83.0763,Y 103.6335,Z 157,A 125.7853,B 20.8127,C -0.8766,E1 20.7314,E2 322.0612} C_DIS
LIN {X -79.7408,Y 106.2211,Z 157,A 123.9334,B 20.8126,C -0.8791,E1 20.7355,E2 323.9143} C_DIS
LIN {X -76.2609,Y 108.7465,Z 157,A 122.0591,B 20.8125,C -0.882,E1 20.7398,E2 325.7885} C_DIS
LIN {X -72.7293,Y 111.1395,Z 157,A 120.2334,B 20.8123,C -0.886,E1 20.744,E2 327.61} C_DIS
LIN {X -69.1798,Y 113.3828,Z 157,A 118.4293,B 20.8122,C -0.8896,E1 20.7483,E2 329.411} C_DIS
LIN {X -65.4787,Y 115.5599,Z 157,A 116.5576,B 20.8121,C -0.892,E1 20.7528,E2 331.2828} C_DIS
LIN {X -62.0539,Y 117.4321,Z 157,A 115.1219,B 20.8115,C -0.9049,E1 20.7562,E2 332.6871} C_DIS
LIN {X -57.8153,Y 119.577,Z 157,A 112.8165,B 20.8118,C -0.8976,E1 20.7621,E2 335.0205} C_DIS
LIN {X -54.5679,Y 121.0924,Z 157,A 111.3284,B 20.8116,C -0.9022,E1 20.7658,E2 336.5} C_DIS
LIN {X -48.6262,Y 123.5989,Z 157,A 108.4868,B 20.8116,C -0.9035,E1 20.7732,E2 339.3457} C_DIS
LIN {X -45.251,Y 124.8731,Z 157,A 107.0152,B 20.8114,C -0.909,E1 20.777,E2 340.8058} C_DIS
LIN {X -42.0624,Y 125.9829,Z 157,A 105.5799,B 20.8113,C -0.9115,E1 20.7808,E2 342.2372} C_DIS
LIN {X -39.528,Y 126.8028,Z 157,A 103.8241,B 20.8122,C -0.8879,E1 20.7857,E2 344.0634} C_DIS
LIN {X -35.113,Y 128.0956,Z 157,A 102.2863,B 20.8114,C -0.9082,E1 20.7896,E2 345.5469} C_DIS
LIN {X -31.9908,Y 128.9109,Z 157,A 100.2645,B 20.8124,C -0.8836,E1 20.7953,E2 347.6415} C_DIS
LIN {X -26.7001,Y 130.1081,Z 157,A 98.6256,B 20.8111,C -0.9143,E1 20.7996,E2 349.1962} C_DIS
LIN {X -21.5617,Y 131.0579,Z 157,A 96.29,B 20.8112,C -0.9125,E1 20.806,E2 351.5397} C_DIS
LIN {X -17.3865,Y 131.6765,Z 157,A 94.6041,B 20.8109,C -0.9192,E1 20.8106,E2 353.2083} C_DIS
LIN {X -14.0391,Y 132.0755,Z 157,A 93.0255,B 20.8111,C -0.9148,E1 20.815,E2 354.8006} C_DIS
LIN {X -9.819,Y 132.4561,Z 157,A 91.2799,B 20.8109,C -0.919,E1 20.8199,E2 356.5354} C_DIS
LIN {X -6.1514,Y 132.678,Z 157,A 89.5821,B 20.8111,C -0.9147,E1 20.8246,E2 358.2457} C_DIS
LIN {X -2.0757,Y 132.8034,Z 157,A 87.9187,B 20.8109,C -0.9192,E1 20.8292,E2 359.8968} C_DIS
LIN {X 2.0855,Y 132.8032,Z 157,A 86.1454,B 20.8109,C -0.9203,E1 20.8342,E2 361.6666} C_DIS
LIN {X 5.7908,Y 132.6947,Z 157,A 84.4273,B 20.8111,C -0.9153,E1 20.839,E2 363.3982} C_DIS
LIN {X 9.8519,Y 132.4537,Z 157,A 82.7203,B 20.8111,C -0.9173,E1 20.8438,E2 365.0988} C_DIS
LIN {X 14.0504,Y 132.0743,Z 157,A 81.0205,B 20.8108,C -0.9221,E1 20.8484,E2 366.7838} C_DIS
LIN {X 16.5714,Y 131.7834,Z 157,A 79.7652,B 20.8111,C -0.9149,E1 20.852,E2 368.058} C_DIS
LIN {X 20.3231,Y 131.2553,Z 157,A 78.2272,B 20.811,C -0.9186,E1 20.8562,E2 369.5841} C_DIS
LIN {X 24.3448,Y 130.5705,Z 157,A 76.5614,B 20.8108,C -0.9219,E1 20.8607,E2 371.2384} C_DIS
LIN {X 27.6432,Y 129.9114,Z 157,A 74.9915,B 20.8111,C -0.9161,E1 20.8651,E2 372.8222} C_DIS
LIN {X 30.3711,Y 129.3019,Z 157,A 73.5538,B 20.8115,C -0.9054,E1 20.8691,E2 374.2873} C_DIS
LIN {X 33.4798,Y 128.5326,Z 157,A 72.379,B 20.8112,C -0.9134,E1 20.8722,E2 375.4375} C_DIS
LIN {X 38.5664,Y 127.0971,Z 157,A 70.1767,B 20.8112,C -0.9151,E1 20.8781,E2 377.6304} C_DIS
LIN {X 41.7061,Y 126.1015,Z 157,A 68.7747,B 20.8112,C -0.9148,E1 20.8818,E2 379.0302} C_DIS
LIN {X 44.8722,Y 125.0097,Z 157,A 67.3459,B 20.8112,C -0.9141,E1 20.8855,E2 380.4572} C_DIS
LIN {X 47.9092,Y 123.8776,Z 157,A 65.8961,B 20.8113,C -0.9105,E1 20.8893,E2 381.9133} C_DIS
LIN {X 51.3263,Y 122.5012,Z 157,A 64.4106,B 20.8112,C -0.9134,E1 20.8931,E2 383.3866} C_DIS
LIN {X 54.2477,Y 121.2356,Z 157,A 62.9608,B 20.8114,C -0.9085,E1 20.8969,E2 384.8458} C_DIS
LIN {X 57.4725,Y 119.7408,Z 157,A 61.3945,B 20.8115,C -0.9052,E1 20.9008,E2 386.4164} C_DIS
LIN {X 61.4207,Y 117.7646,Z 157,A 59.5352,B 20.8115,C -0.9047,E1 20.9054,E2 388.2708} C_DIS
LIN {X 65.1776,Y 115.7294,Z 157,A 57.633,B 20.8118,C -0.8995,E1 20.9101,E2 390.1807} C_DIS
LIN {X 69.0334,Y 113.4721,Z 157,A 55.6864,B 20.8119,C -0.8958,E1 20.9148,E2 392.1305} C_DIS
LIN {X 72.6022,Y 111.2224,Z 157,A 53.8831,B 20.812,C -0.8936,E1 20.919,E2 393.9326} C_DIS
LIN {X 76.2512,Y 108.7534,Z 157,A 51.9455,B 20.8122,C -0.8888,E1 20.9235,E2 395.8756} C_DIS
LIN {X 79.1609,Y 106.6537,Z 157,A 50.4284,B 20.8122,C -0.8875,E1 20.9269,E2 397.3898} C_DIS
LIN {X 82.8368,Y 103.8243,Z 157,A 48.7339,B 20.8118,C -0.8975,E1 20.9306,E2 399.0485} C_DIS
LIN {X 85.9162,Y 101.2908,Z 157,A 46.7417,B 20.8125,C -0.8821,E1 20.9349,E2 401.0746} C_DIS
LIN {X 88.7793,Y 98.7911,Z 157,A 44.6272,B 20.8134,C -0.8577,E1 20.9395,E2 403.2471} C_DIS
LIN {X 92.2254,Y 95.582,Z 157,A 43.075,B 20.8128,C -0.8748,E1 20.9425,E2 404.7435} C_DIS
LIN {X 95.4174,Y 92.3955,Z 157,A 41.1735,B 20.8128,C -0.8726,E1 20.9462,E2 406.6413} C_DIS
LIN {X 97.8158,Y 89.8525,Z 157,A 39.477,B 20.8133,C -0.8608,E1 20.9494,E2 408.3616} C_DIS
LIN {X 101.388,Y 85.8019,Z 157,A 36.9419,B 20.8139,C -0.8462,E1 20.9541,E2 410.9234} C_DIS
LIN {X 104.0825,Y 82.5125,Z 157,A 35.5265,B 20.8133,C -0.8607,E1 20.9565,E2 412.2902} C_DIS
LIN {X 106.7738,Y 78.9995,Z 157,A 33.7114,B 20.8133,C -0.8603,E1 20.9595,E2 414.0958} C_DIS
LIN {X 109.0408,Y 75.8387,Z 157,A 31.9854,B 20.8136,C -0.8539,E1 20.9623,E2 415.8293} C_DIS
LIN {X 111.3336,Y 72.431,Z 157,A 30.1794,B 20.8138,C -0.8478,E1 20.9651,E2 417.6414} C_DIS
LIN {X 113.6922,Y 68.6695,Z 157,A 28.3392,B 20.8138,C -0.8462,E1 20.9678,E2 419.4746} C_DIS
LIN {X 115.7894,Y 65.0709,Z 157,A 26.5156,B 20.8141,C -0.8402,E1 20.9703,E2 421.3035} C_DIS
LIN {X 117.9856,Y 60.9998,Z 157,A 24.6191,B 20.8141,C -0.8393,E1 20.9728,E2 423.1903} C_DIS
LIN {X 119.6503,Y 57.6618,Z 157,A 22.9517,B 20.8144,C -0.8322,E1 20.9749,E2 424.8666} C_DIS
LIN {X 121.219,Y 54.2848,Z 157,A 21.4373,B 20.8144,C -0.8319,E1 20.9766,E2 426.3719} C_DIS
LIN {X 122.5099,Y 51.3054,Z 157,A 20.0407,B 20.8146,C -0.828,E1 20.9781,E2 427.7697} C_DIS
LIN {X 123.7822,Y 48.1546,Z 157,A 18.5888,B 20.8147,C -0.8244,E1 20.9796,E2 429.2219} C_DIS
LIN {X 124.9567,Y 45.0193,Z 157,A 17.1124,B 20.8149,C -0.8188,E1 20.9811,E2 430.704} C_DIS
LIN {X 126.294,Y 41.1255,Z 157,A 15.4174,B 20.815,C -0.8172,E1 20.9826,E2 432.3917} C_DIS
LIN {X 127.77,Y 36.2771,Z 157,A 13.148,B 20.8154,C -0.8068,E1 20.9844,E2 434.6742} C_DIS
LIN {X 128.7295,Y 32.7058,Z 157,A 11.6062,B 20.8154,C -0.8045,E1 20.9855,E2 436.2117} C_DIS
LIN {X 130.2036,Y 26.2308,Z 157,A 8.6746,B 20.8159,C -0.7926,E1 20.9872,E2 439.1556} C_DIS
LIN {X 130.9797,Y 22.0303,Z 157,A 6.9449,B 20.8159,C -0.7921,E1 20.9881,E2 440.8744} C_DIS
LIN {X 131.4486,Y 19.0342,Z 157,A 5.6397,B 20.8161,C -0.7882,E1 20.9886,E2 442.1811} C_DIS
LIN {X 131.9014,Y 15.5897,Z 157,A 4.1281,B 20.8163,C -0.7829,E1 20.9891,E2 443.6966} C_DIS
LIN {X 132.3354,Y 11.3306,Z 157,A 2.3545,B 20.8163,C -0.7804,E1 20.9896,E2 445.4641} C_DIS
LIN {X 132.5801,Y 7.9726,Z 157,A 0.8431,B 20.8166,C -0.7731,E1 20.9899,E2 446.985} C_DIS
LIN {X 132.7624,Y 3.9022,Z 157,A -0.8776,B 20.8168,C -0.7693,E1 20.9901,E2 448.7039} C_DIS
LIN {X 132.822,Y -0.1688,Z 157,A -2.7388,B 20.8171,C -0.7588,E1 20.9901,E2 450.5808} C_DIS
LIN {X 132.7431,Y -4.5477,Z 157,A -4.5628,B 20.8172,C -0.7558,E1 20.99,E2 452.3998} C_DIS
LIN {X 132.5733,Y -8.0831,Z 157,A -5.9863,B 20.8172,C -0.7558,E1 20.9898,E2 453.8131} C_DIS
LIN {X 132.3129,Y -11.5971,Z 157,A -7.7296,B 20.8177,C -0.7406,E1 20.9894,E2 455.5862} C_DIS
LIN {X 131.7907,Y -16.5157,Z 157,A -9.7317,B 20.8177,C -0.7399,E1 20.9887,E2 457.5758} C_DIS
LIN {X 131.3135,Y -19.9472,Z 157,A -11.1095,B 20.8177,C -0.7406,E1 20.9882,E2 458.9418} C_DIS
LIN {X 130.6081,Y -24.147,Z 157,A -13.0362,B 20.8181,C -0.7306,E1 20.9872,E2 460.8824} C_DIS
LIN {X 129.9774,Y -27.3375,Z 157,A -14.5575,B 20.8184,C -0.7207,E1 20.9864,E2 462.4205} C_DIS
LIN {X 128.8242,Y -32.3324,Z 157,A -16.5345,B 20.8183,C -0.7246,E1 20.9851,E2 464.3726} C_DIS
LIN {X 127.8993,Y -35.8148,Z 157,A -17.9486,B 20.8183,C -0.7263,E1 20.9841,E2 465.772} C_DIS
LIN {X 126.4035,Y -40.7826,Z 157,A -20.372,B 20.8187,C -0.7108,E1 20.982,E2 468.2219} C_DIS
LIN {X 125.1289,Y -44.5418,Z 157,A -22.0151,B 20.8188,C -0.7087,E1 20.9805,E2 469.8594} C_DIS
LIN {X 123.2063,Y -49.6096,Z 157,A -24.2756,B 20.8189,C -0.7053,E1 20.9783,E2 472.1143} C_DIS
LIN {X 121.8973,Y -52.744,Z 157,A -25.8217,B 20.8192,C -0.6971,E1 20.9766,E2 473.6727} C_DIS
LIN {X 119.974,Y -56.9843,Z 157,A -27.6657,B 20.8192,C -0.6988,E1 20.9744,E2 475.4998} C_DIS
LIN {X 118.6014,Y -59.7901,Z 157,A -29.1825,B 20.8195,C -0.687,E1 20.9725,E2 477.0397} C_DIS
LIN {X 116.7351,Y -63.3593,Z 157,A -30.9014,B 20.8196,C -0.6828,E1 20.9702,E2 478.7592} C_DIS
LIN {X 114.6116,Y -67.1239,Z 157,A -32.7443,B 20.8198,C -0.6785,E1 20.9677,E2 480.6025} C_DIS
LIN {X 112.3025,Y -70.9193,Z 157,A -34.6361,B 20.8198,C -0.6743,E1 20.9649,E2 482.4944} C_DIS
LIN {X 109.5298,Y -75.1307,Z 157,A -37.3694,B 20.8208,C -0.6428,E1 20.9605,E2 485.2991} C_DIS
LIN {X 106.5272,Y -79.3306,Z 157,A -38.9843,B 20.8202,C -0.6648,E1 20.958,E2 486.843} C_DIS
LIN {X 104.0828,Y -82.512,Z 157,A -40.75,B 20.8204,C -0.6587,E1 20.9549,E2 488.6157} C_DIS
LIN {X 101.2982,Y -85.9075,Z 157,A -42.6211,B 20.8204,C -0.6549,E1 20.9516,E2 490.4869} C_DIS
LIN {X 99.4702,Y -88.0176,Z 157,A -44.0379,B 20.8209,C -0.6421,E1 20.9489,E2 491.9315} C_DIS
LIN {X 97.2045,Y -90.5135,Z 157,A -45.4142,B 20.8209,C -0.6421,E1 20.9463,E2 493.3005} C_DIS
LIN {X 93.4571,Y -94.378,Z 157,A -47.5149,B 20.8207,C -0.6466,E1 20.9422,E2 495.3776} C_DIS
LIN {X 90.3929,Y -97.3168,Z 157,A -49.1834,B 20.8207,C -0.6498,E1 20.9389,E2 497.0287} C_DIS
LIN {X 87.9655,Y -99.5162,Z 157,A -50.9851,B 20.8213,C -0.6289,E1 20.935,E2 498.8801} C_DIS
LIN {X 85.5303,Y -101.617,Z 157,A -52.1906,B 20.8211,C -0.6341,E1 20.9325,E2 500.0653} C_DIS
LIN {X 81.9838,Y -104.4991,Z 157,A -54.1003,B 20.8211,C -0.6327,E1 20.9283,E2 501.9702} C_DIS
LIN {X 78.0759,Y -107.4504,Z 157,A -56.4327,B 20.8216,C -0.6185,E1 20.923,E2 504.3323} C_DIS
LIN {X 75.4217,Y -109.3301,Z 157,A -57.5816,B 20.8213,C -0.6271,E1 20.9205,E2 505.4521} C_DIS
LIN {X 72.5623,Y -111.2483,Z 157,A -60.0032,B 20.8225,C -0.5824,E1 20.9145,E2 507.9892} C_DIS
LIN {X 66.726,Y -114.8438,Z 157,A -62.0458,B 20.8216,C -0.6179,E1 20.9099,E2 509.9246} C_DIS
LIN {X 62.9028,Y -116.9814,Z 157,A -63.8237,B 20.8216,C -0.6197,E1 20.9055,E2 511.6912} C_DIS
LIN {X 59.3604,Y -118.8178,Z 157,A -65.7151,B 20.8218,C -0.6093,E1 20.9008,E2 513.6054} C_DIS
LIN {X 55.5777,Y -120.6318,Z 157,A -67.3418,B 20.8217,C -0.6147,E1 20.8967,E2 515.2118} C_DIS
LIN {X 52.6072,Y -121.9565,Z 157,A -68.6647,B 20.8217,C -0.6163,E1 20.8934,E2 516.5264} C_DIS
LIN {X 49.7101,Y -123.1658,Z 157,A -70.1407,B 20.8218,C -0.6089,E1 20.8895,E2 518.0187} C_DIS
LIN {X 45.9132,Y -124.6331,Z 157,A -71.9918,B 20.822,C -0.6024,E1 20.8846,E2 519.8833} C_DIS
LIN {X 42.1324,Y -125.9596,Z 157,A -73.6882,B 20.822,C -0.6017,E1 20.8802,E2 521.5774} C_DIS
LIN {X 37.8894,Y -127.3015,Z 157,A -75.5117,B 20.822,C -0.6038,E1 20.8753,E2 523.3911} C_DIS
LIN {X 34.628,Y -128.2264,Z 157,A -76.9719,B 20.822,C -0.6024,E1 20.8714,E2 524.8524} C_DIS
LIN {X 31.2631,Y -129.0875,Z 157,A -78.4432,B 20.822,C -0.6022,E1 20.8674,E2 526.3215} C_DIS
LIN {X 28.0101,Y -129.8322,Z 157,A -79.9384,B 20.8221,C -0.5985,E1 20.8633,E2 527.8248} C_DIS
LIN {X 23.2001,Y -130.7775,Z 157,A -82.0026,B 20.8221,C -0.599,E1 20.8577,E2 529.8845} C_DIS
LIN {X 19.1957,Y -131.4256,Z 157,A -83.807,B 20.8221,C -0.5954,E1 20.8527,E2 531.6969} C_DIS
LIN {X 15.4502,Y -131.918,Z 157,A -85.3903,B 20.8221,C -0.5965,E1 20.8483,E2 533.2757} C_DIS
LIN {X 11.4271,Y -132.3272,Z 157,A -87.1525,B 20.8222,C -0.5948,E1 20.8434,E2 535.0411} C_DIS
LIN {X 7.5579,Y -132.6057,Z 157,A -88.8972,B 20.8223,C -0.5911,E1 20.8385,E2 536.7956} C_DIS
LIN {X 3.6382,Y -132.7697,Z 157,A -90.4969,B 20.8223,C -0.5946,E1 20.834,E2 538.3849} C_DIS
LIN {X 0.9345,Y -132.8131,Z 157,A -91.4854,B 20.822,C -0.6021,E1 20.8313,E2 539.3521} C_DIS
Enddeposition()
LIN {X 0.9345,Y -132.8131,Z 157,A -91.4854,B 20.822,C -0.6021,E1 20.8313,E2 539.3521} C_DIS
Startdeposition()
$VEL.CP = VEL_PRINT
LIN {X 2.3218,Y -131.8677,Z 157,A -90.0153,B 19.6628,C -0.4764,E1 19.6727,E2 538.1331} C_DIS
LIN {X 6.3865,Y -131.7335,Z 157,A -88.2298,B 19.6628,C -0.4777,E1 19.6777,E2 536.3443} C_DIS
LIN {X 9.8152,Y -131.5224,Z 157,A -86.7665,B 19.6628,C -0.4771,E1 19.6818,E2 534.8837} C_DIS
LIN {X 13.8976,Y -131.1538,Z 157,A -84.9847,B 19.6628,C -0.478,E1 19.6867,E2 533.1005} C_DIS
LIN {X 17.2597,Y -130.7537,Z 157,A -83.4936,B 19.6628,C -0.4797,E1 19.6909,E2 531.6059} C_DIS
LIN {X 22.1647,Y -130.0129,Z 157,A -81.3953,B 19.6628,C -0.4788,E1 19.6966,E2 529.513} C_DIS
LIN {X 28.2585,Y -128.8256,Z 157,A -78.7475,B 19.6628,C -0.4788,E1 19.7039,E2 526.8693} C_DIS
LIN {X 31.038,Y -128.1836,Z 157,A -77.4445,B 19.6626,C -0.4827,E1 19.7074,E2 525.5574} C_DIS
LIN {X 35.0053,Y -127.1585,Z 157,A -75.3658,B 19.6623,C -0.497,E1 19.7132,E2 523.4405} C_DIS
LIN {X 38.1612,Y -126.2469,Z 157,A -73.8309,B 19.6621,C -0.5032,E1 19.7173,E2 521.891} C_DIS
LIN {X 41.8233,Y -125.0807,Z 157,A -72.5585,B 19.6625,C -0.4883,E1 19.7205,E2 520.6659} C_DIS
LIN {X 45.7447,Y -123.7015,Z 157,A -70.7198,B 19.6625,C -0.4919,E1 19.7254,E2 518.8214} C_DIS
LIN {X 49.5441,Y -122.2284,Z 157,A -69.063,B 19.6625,C -0.4895,E1 19.7297,E2 517.1767} C_DIS
LIN {X 52.4518,Y -121.0089,Z 157,A -67.6758,B 19.6625,C -0.4921,E1 19.7332,E2 515.786} C_DIS
LIN {X 55.7256,Y -119.5372,Z 157,A -66.0858,B 19.6623,C -0.4957,E1 19.7373,E2 514.1905} C_DIS
LIN {X 62.2982,Y -116.2488,Z 157,A -63.1531,B 19.6625,C -0.4897,E1 19.7445,E2 511.2862} C_DIS
LIN {X 64.8232,Y -114.86,Z 157,A -61.5933,B 19.6621,C -0.5049,E1 19.7484,E2 509.6873} C_DIS
LIN {X 69.1186,Y -112.3269,Z 157,A -59.1215,B 19.6617,C -0.5219,E1 19.7544,E2 507.1752} C_DIS
LIN {X 72.3528,Y -110.2721,Z 157,A -58.011,B 19.6622,C -0.5012,E1 19.7569,E2 506.1308} C_DIS
LIN {X 74.7526,Y -108.6595,Z 157,A -56.541,B 19.6619,C -0.5128,E1 19.7603,E2 504.633} C_DIS
LIN {X 79.6006,Y -105.1599,Z 157,A -53.3936,B 19.6612,C -0.5419,E1 19.7675,E2 501.4142} C_DIS
LIN {X 83.5491,Y -102.0509,Z 157,A -52.1159,B 19.662,C -0.5072,E1 19.7701,E2 500.2452} C_DIS
LIN {X 88.3217,Y -97.9503,Z 157,A -48.6026,B 19.661,C -0.547,E1 19.7777,E2 496.6323} C_DIS
LIN {X 91.605,Y -94.8862,Z 157,A -47.3958,B 19.6617,C -0.5192,E1 19.7799,E2 495.5145} C_DIS
LIN {X 93.7909,Y -92.7265,Z 157,A -45.195,B 19.6607,C -0.56,E1 19.7845,E2 493.2051} C_DIS
LIN {X 97.4175,Y -88.9089,Z 157,A -42.9106,B 19.6605,C -0.5655,E1 19.7888,E2 490.9177} C_DIS
LIN {X 100.9095,Y -84.9243,Z 157,A -41.3855,B 19.6613,C -0.5372,E1 19.7914,E2 489.4852} C_DIS
LIN {X 102.9036,Y -82.4975,Z 157,A -39.5292,B 19.6606,C -0.5622,E1 19.7947,E2 487.5662} C_DIS
LIN {X 105.3122,Y -79.3987,Z 157,A -37.9259,B 19.6606,C -0.5622,E1 19.7974,E2 485.973} C_DIS
LIN {X 107.3819,Y -76.5766,Z 157,A -36.7114,B 19.6609,C -0.5529,E1 19.7993,E2 484.7938} C_DIS
LIN {X 109.2013,Y -73.9588,Z 157,A -35.3115,B 19.6607,C -0.5573,E1 19.8015,E2 483.39} C_DIS
LIN {X 111.5896,Y -70.3037,Z 157,A -33.4313,B 19.6607,C -0.5617,E1 19.8044,E2 481.5089} C_DIS
LIN {X 113.8072,Y -66.6542,Z 157,A -31.5727,B 19.6605,C -0.5671,E1 19.807,E2 479.647} C_DIS
LIN {X 115.9796,Y -62.7991,Z 157,A -29.6006,B 19.6603,C -0.5747,E1 19.8097,E2 477.6658} C_DIS
LIN {X 118.7453,Y -57.3953,Z 157,A -27.2313,B 19.6603,C -0.5705,E1 19.8126,E2 475.3252} C_DIS
LIN {X 120.5673,Y -53.4605,Z 157,A -25.1426,B 19.66,C -0.5851,E1 19.8151,E2 473.2083} C_DIS
LIN {X 123.6001,Y -46.0154,Z 157,A -21.8434,B 19.66,C -0.5869,E1 19.8185,E2 469.9274} C_DIS
LIN {X 124.6465,Y -43.1,Z 157,A -20.4482,B 19.6597,C -0.5932,E1 19.8198,E2 468.524} C_DIS
LIN {X 125.9008,Y -39.2922,Z 157,A -17.857,B 19.6584,C -0.6362,E1 19.822,E2 465.8251} C_DIS
LIN {X 127.6342,Y -33.2337,Z 157,A -16.0436,B 19.6594,C -0.6035,E1 19.8233,E2 464.1216} C_DIS
LIN {X 129.2288,Y -26.3497,Z 157,A -12.9664,B 19.6591,C -0.6134,E1 19.8252,E2 461.0387} C_DIS
LIN {X 130.2025,Y -21.028,Z 157,A -10.701,B 19.6591,C -0.6169,E1 19.8262,E2 458.7801} C_DIS
LIN {X 130.801,Y -16.8984,Z 157,A -8.8691,B 19.6588,C -0.6235,E1 19.8269,E2 456.9429} C_DIS
LIN {X 131.4863,Y -10.3102,Z 157,A -6.0472,B 19.6586,C -0.63,E1 19.8277,E2 454.1235} C_DIS
LIN {X 131.7688,Y -5.6276,Z 157,A -3.8917,B 19.6583,C -0.6416,E1 19.828,E2 451.9505} C_DIS
LIN {X 131.8762,Y -1.8116,Z 157,A -2.2447,B 19.6581,C -0.6463,E1 19.8281,E2 450.3023} C_DIS
LIN {X 131.8661,Y 2.4157,Z 157,A -0.5388,B 19.6581,C -0.6463,E1 19.8281,E2 448.6096} C_DIS
LIN {X 131.7607,Y 5.8354,Z 157,A 1.0924,B 19.6578,C -0.6574,E1 19.8279,E2 446.9585} C_DIS
LIN {X 131.5277,Y 9.7428,Z 157,A 2.6856,B 19.6578,C -0.658,E1 19.8276,E2 445.3759} C_DIS
LIN {X 131.1443,Y 13.9864,Z 157,A 4.5038,B 19.6576,C -0.6623,E1 19.8271,E2 443.5589} C_DIS
LIN {X 130.7152,Y 17.5537,Z 157,A 6.1817,B 19.6573,C -0.6723,E1 19.8265,E2 441.8645} C_DIS
LIN {X 130.1212,Y 21.5151,Z 157,A 7.779,B 19.6573,C -0.6713,E1 19.8258,E2 440.2822} C_DIS
LIN {X 129.039,Y 27.2689,Z 157,A 11.0362,B 19.656,C -0.7106,E1 19.824,E2 436.9339} C_DIS
LIN {X 127.776,Y 32.6759,Z 157,A 12.7054,B 19.6569,C -0.685,E1 19.8229,E2 435.3526} C_DIS
LIN {X 126.5661,Y 37.086,Z 157,A 14.8546,B 19.6564,C -0.6981,E1 19.8212,E2 433.181} C_DIS
LIN {X 125.3832,Y 40.9148,Z 157,A 16.5345,B 19.6564,C -0.7005,E1 19.8198,E2 431.5064} C_DIS
LIN {X 124.0639,Y 44.7492,Z 157,A 18.1797,B 19.6564,C -0.7005,E1 19.8183,E2 429.873} C_DIS
LIN {X 122.8167,Y 48.0675,Z 157,A 19.6551,B 19.6563,C -0.7022,E1 19.8168,E2 428.4036} C_DIS
LIN {X 121.6669,Y 50.9068,Z 157,A 21.0008,B 19.6561,C -0.7066,E1 19.8154,E2 427.0544} C_DIS
LIN {X 120.321,Y 54.0112,Z 157,A 22.4698,B 19.656,C -0.7107,E1 19.8137,E2 425.5839} C_DIS
LIN {X 118.8626,Y 57.1499,Z 157,A 23.9206,B 19.656,C -0.7126,E1 19.812,E2 424.1376} C_DIS
LIN {X 116.8363,Y 61.1851,Z 157,A 25.6062,B 19.6562,C -0.7059,E1 19.8099,E2 422.4833} C_DIS
LIN {X 115.5659,Y 63.557,Z 157,A 27.0784,B 19.6556,C -0.7222,E1 19.8079,E2 420.9732} C_DIS
LIN {X 113.4867,Y 67.1992,Z 157,A 28.916,B 19.6554,C -0.7277,E1 19.8053,E2 419.1317} C_DIS
LIN {X 111.2775,Y 70.7975,Z 157,A 30.7941,B 19.6552,C -0.7343,E1 19.8025,E2 417.2465} C_DIS
LIN {X 108.8996,Y 74.4028,Z 157,A 32.8465,B 19.6547,C -0.7466,E1 19.7993,E2 415.1709} C_DIS
LIN {X 106.9812,Y 77.136,Z 157,A 34.0329,B 19.655,C -0.7388,E1 19.7974,E2 414.0152} C_DIS
LIN {X 104.5078,Y 80.4557,Z 157,A 35.8918,B 19.6547,C -0.7457,E1 19.7942,E2 412.1474} C_DIS
LIN {X 101.0102,Y 84.8042,Z 157,A 38.2177,B 19.6547,C -0.7471,E1 19.7901,E2 409.8312} C_DIS
LIN {X 99.1681,Y 86.9518,Z 157,A 39.5031,B 19.6545,C -0.7523,E1 19.7878,E2 408.5381} C_DIS
LIN {X 96.196,Y 90.2292,Z 157,A 41.4346,B 19.6543,C -0.757,E1 19.7841,E2 406.604} C_DIS
LIN {X 93.1007,Y 93.4191,Z 157,A 43.3362,B 19.6543,C -0.7598,E1 19.7804,E2 404.7045} C_DIS
LIN {X 88.2449,Y 98.0181,Z 157,A 46.2147,B 19.6541,C -0.7645,E1 19.7745,E2 401.8273} C_DIS
LIN {X 86.0311,Y 99.9674,Z 157,A 47.5134,B 19.6539,C -0.7677,E1 19.7717,E2 400.5257} C_DIS
LIN {X 82.4483,Y 102.943,Z 157,A 49.3907,B 19.654,C -0.7653,E1 19.7677,E2 398.6649} C_DIS
LIN {X 79.4022,Y 105.3096,Z 157,A 51.1546,B 19.6538,C -0.7721,E1 19.7638,E2 396.8894} C_DIS
LIN {X 75.7383,Y 107.9752,Z 157,A 53.1394,B 19.6536,C -0.7761,E1 19.7592,E2 394.9017} C_DIS
LIN {X 72.1543,Y 110.4026,Z 157,A 55.0183,B 19.6536,C -0.7791,E1 19.7549,E2 393.0223} C_DIS
LIN {X 68.4629,Y 112.7285,Z 157,A 56.899,B 19.6534,C -0.7813,E1 19.7504,E2 391.1427} C_DIS
LIN {X 64.4525,Y 115.0684,Z 157,A 58.8398,B 19.6534,C -0.781,E1 19.7457,E2 389.2103} C_DIS
LIN {X 61.1656,Y 116.8465,Z 157,A 60.3672,B 19.6534,C -0.7792,E1 19.742,E2 387.6939} C_DIS
LIN {X 58.274,Y 118.315,Z 157,A 61.8086,B 19.6534,C -0.7824,E1 19.7384,E2 386.2483} C_DIS
LIN {X 54.9991,Y 119.8731,Z 157,A 63.3548,B 19.6534,C -0.7831,E1 19.7345,E2 384.7053} C_DIS
LIN {X 52.1152,Y 121.1544,Z 157,A 64.8386,B 19.6531,C -0.7893,E1 19.7306,E2 383.2078} C_DIS
LIN {X 47.7859,Y 122.9261,Z 157,A 66.816,B 19.6531,C -0.7891,E1 19.7255,E2 381.2367} C_DIS
LIN {X 44.2903,Y 124.2293,Z 157,A 68.3668,B 19.6531,C -0.7877,E1 19.7215,E2 379.6942} C_DIS
LIN {X 41.4217,Y 125.2144,Z 157,A 69.6885,B 19.6531,C -0.789,E1 19.718,E2 378.3719} C_DIS
LIN {X 38.0806,Y 126.2716,Z 157,A 71.5536,B 19.6525,C -0.8043,E1 19.7129,E2 376.4659} C_DIS
LIN {X 34.8563,Y 127.1995,Z 157,A 72.6435,B 19.6531,C -0.7902,E1 19.7101,E2 375.4202} C_DIS
LIN {X 31.7254,Y 128.0172,Z 157,A 74.408,B 19.6525,C -0.8058,E1 19.7052,E2 373.6129} C_DIS
LIN {X 28.5828,Y 128.7542,Z 157,A 75.5532,B 19.6529,C -0.7961,E1 19.7022,E2 372.4986} C_DIS
LIN {X 24.8251,Y 129.5303,Z 157,A 77.1654,B 19.6529,C -0.7946,E1 19.6978,E2 370.8933} C_DIS
LIN {X 21.2553,Y 130.1646,Z 157,A 78.8031,B 19.6528,C -0.7978,E1 19.6932,E2 369.2485} C_DIS
LIN {X 15.8469,Y 130.9326,Z 157,A 80.8621,B 19.6533,C -0.7857,E1 19.6876,E2 367.2275} C_DIS
LIN {X 11.3037,Y 131.4028,Z 157,A 83.0932,B 19.6529,C -0.796,E1 19.6814,E2 364.9678} C_DIS
LIN {X 7.7901,Y 131.6581,Z 157,A 84.7359,B 19.6527,C -0.8006,E1 19.6767,E2 363.3123} C_DIS
LIN {X 3.6119,Y 131.8386,Z 157,A 86.4188,B 19.6529,C -0.7952,E1 19.6721,E2 361.6461} C_DIS
LIN {X 0.0504,Y 131.8898,Z 157,A 88.1002,B 19.6527,C -0.8003,E1 19.6674,E2 359.9496} C_DIS
LIN {X -3.8364,Y 131.8323,Z 157,A 89.6959,B 19.6528,C -0.7963,E1 19.6629,E2 358.3658} C_DIS
LIN {X -8.004,Y 131.6449,Z 157,A 91.5069,B 19.6528,C -0.7957,E1 19.6579,E2 356.556} C_DIS
LIN {X -11.9001,Y 131.3519,Z 157,A 93.6933,B 19.6521,C -0.8144,E1 19.6517,E2 354.3123} C_DIS
LIN {X -16.1313,Y 130.8987,Z 157,A 94.9799,B 19.653,C -0.7911,E1 19.6483,E2 353.094} C_DIS
LIN {X -18.8952,Y 130.5275,Z 157,A 96.3003,B 19.653,C -0.7948,E1 19.6446,E2 351.7614} C_DIS
LIN {X -25.9295,Y 129.3143,Z 157,A 99.173,B 19.6533,C -0.7836,E1 19.6368,E2 348.9183} C_DIS
LIN {X -31.2824,Y 128.1247,Z 157,A 101.9444,B 19.6528,C -0.7968,E1 19.6291,E2 346.1027} C_DIS
LIN {X -35.1752,Y 127.111,Z 157,A 103.6573,B 19.6529,C -0.7938,E1 19.6245,E2 344.3954} C_DIS
LIN {X -40.7147,Y 125.4473,Z 157,A 105.9575,B 19.6534,C -0.7828,E1 19.6184,E2 342.1228} C_DIS
LIN {X -43.5924,Y 124.4758,Z 157,A 107.3184,B 19.6534,C -0.7829,E1 19.6148,E2 340.7583} C_DIS
LIN {X -46.5888,Y 123.3853,Z 157,A 108.8152,B 19.6533,C -0.7855,E1 19.6109,E2 339.2497} C_DIS
LIN {X -55.0301,Y 119.8588,Z 157,A 112.5599,B 19.6538,C -0.7712,E1 19.6014,E2 335.5364} C_DIS
LIN {X -57.7065,Y 118.595,Z 157,A 114.6268,B 19.6527,C -0.7995,E1 19.5959,E2 333.3782} C_DIS
LIN {X -62.0655,Y 116.3737,Z 157,A 116.2429,B 19.6536,C -0.7763,E1 19.5921,E2 331.8253} C_DIS
LIN {X -65.8214,Y 114.2911,Z 157,A 118.1432,B 19.6536,C -0.7746,E1 19.5875,E2 329.923} C_DIS
LIN {X -69.6124,Y 112.0221,Z 157,A 120.0311,B 19.6538,C -0.77,E1 19.583,E2 328.0411} C_DIS
LIN {X -73.4384,Y 109.5522,Z 157,A 122.0284,B 19.654,C -0.7671,E1 19.5783,E2 326.0441} C_DIS
LIN {X -77.0576,Y 107.038,Z 157,A 123.9932,B 19.654,C -0.7653,E1 19.5738,E2 324.0758} C_DIS
LIN {X -80.6367,Y 104.3676,Z 157,A 125.9188,B 19.6542,C -0.7608,E1 19.5696,E2 322.1544} C_DIS
LIN {X -84.2289,Y 101.4906,Z 157,A 127.9084,B 19.6544,C -0.7563,E1 19.5653,E2 320.1686} C_DIS
LIN {X -87.667,Y 98.5368,Z 157,A 129.9371,B 19.6544,C -0.7542,E1 19.561,E2 318.1355} C_DIS
LIN {X -90.9833,Y 95.4824,Z 157,A 131.8812,B 19.6546,C -0.7493,E1 19.557,E2 316.1958} C_DIS
LIN {X -94.2141,Y 92.2959,Z 157,A 133.8473,B 19.6548,C -0.7445,E1 19.5532,E2 314.2331} C_DIS
LIN {X -97.2653,Y 89.075,Z 157,A 135.783,B 19.6549,C -0.7402,E1 19.5495,E2 312.2993} C_DIS
LIN {X -100.2086,Y 85.751,Z 157,A 137.7699,B 19.655,C -0.7376,E1 19.5458,E2 310.3083} C_DIS
LIN {X -103.0035,Y 82.3723,Z 157,A 139.682,B 19.6552,C -0.7331,E1 19.5425,E2 308.3981} C_DIS
LIN {X -105.807,Y 78.7382,Z 157,A 141.6519,B 19.6554,C -0.727,E1 19.5392,E2 306.4341} C_DIS
LIN {X -108.4733,Y 75.0234,Z 157,A 143.6578,B 19.6556,C -0.7225,E1 19.5359,E2 304.4289} C_DIS
LIN {X -110.7984,Y 71.5447,Z 157,A 145.4586,B 19.6558,C -0.717,E1 19.5332,E2 302.6329} C_DIS
LIN {X -112.9082,Y 68.1658,Z 157,A 147.1743,B 19.656,C -0.7116,E1 19.5307,E2 300.9217} C_DIS
LIN {X -114.9282,Y 64.702,Z 157,A 149.5136,B 19.6553,C -0.7291,E1 19.5274,E2 298.5139} C_DIS
LIN {X -117.2319,Y 60.427,Z 157,A 151.1435,B 19.6562,C -0.7051,E1 19.5254,E2 296.9445} C_DIS
LIN {X -120.1526,Y 54.3877,Z 157,A 153.8541,B 19.6567,C -0.6891,E1 19.5222,E2 294.2627} C_DIS
LIN {X -121.673,Y 50.8921,Z 157,A 155.6247,B 19.6567,C -0.6885,E1 19.5202,E2 292.4812} C_DIS
LIN {X -123.0408,Y 47.491,Z 157,A 157.21,B 19.6569,C -0.6835,E1 19.5186,E2 290.8993} C_DIS
LIN {X -124.1704,Y 44.4537,Z 157,A 158.6186,B 19.6571,C -0.6793,E1 19.5172,E2 289.4928} C_DIS
LIN {X -125.1858,Y 41.5078,Z 157,A 160.0229,B 19.6571,C -0.6771,E1 19.516,E2 288.0846} C_DIS
LIN {X -126.2367,Y 38.1946,Z 157,A 161.6683,B 19.6571,C -0.6775,E1 19.5146,E2 286.4256} C_DIS
LIN {X -127.4223,Y 34.0283,Z 157,A 163.4134,B 19.6575,C -0.6667,E1 19.5133,E2 284.6997} C_DIS
LIN {X -128.2906,Y 30.5939,Z 157,A 164.9982,B 19.6575,C -0.6636,E1 19.5123,E2 283.1119} C_DIS
LIN {X -129.1896,Y 26.5424,Z 157,A 166.7158,B 19.6579,C -0.6549,E1 19.5113,E2 281.4073} C_DIS
LIN {X -130.3711,Y 19.9461,Z 157,A 169.6597,B 19.6581,C -0.647,E1 19.5099,E2 278.4643} C_DIS
LIN {X -130.8,Y 16.9067,Z 157,A 171.4513,B 19.6577,C -0.6598,E1 19.5092,E2 276.6202} C_DIS
LIN {X -131.2223,Y 13.25,Z 157,A 172.6182,B 19.6584,C -0.6387,E1 19.5089,E2 275.5073} C_DIS
LIN {X -131.5193,Y 9.858,Z 157,A 174.1383,B 19.6584,C -0.6356,E1 19.5085,E2 273.9846} C_DIS
LIN {X -131.7204,Y 6.6476,Z 157,A 175.6101,B 19.6585,C -0.634,E1 19.5083,E2 272.5062} C_DIS
LIN {X -131.8897,Y 0.2919,Z 157,A 178.8034,B 19.6583,C -0.6413,E1 19.5081,E2 269.2657} C_DIS
LIN {X -131.8437,Y -3.4289,Z 157,A 179.7728,B 19.6592,C -0.6123,E1 19.5082,E2 268.3757} C_DIS
LIN {X -131.6377,Y -8.1206,Z 157,A -177.2633,B 19.6583,C -0.6403,E1 19.5087,E2 265.3046} C_DIS
LIN {X -131.2172,Y -13.3027,Z 157,A -175.3969,B 19.659,C -0.6185,E1 19.5091,E2 263.4887} C_DIS
LIN {X -130.3609,Y -20.012,Z 157,A -172.9549,B 19.6598,C -0.591,E1 19.51,E2 261.1101} C_DIS
LIN {X -129.4362,Y -25.3168,Z 157,A -170.0623,B 19.6594,C -0.6044,E1 19.5115,E2 258.1548} C_DIS
LIN {X -128.606,Y -29.2387,Z 157,A -168.5736,B 19.6598,C -0.5897,E1 19.5124,E2 256.6987} C_DIS
LIN {X -127.8283,Y -32.4701,Z 157,A -167.1349,B 19.66,C -0.5852,E1 19.5133,E2 255.2626} C_DIS
LIN {X -126.9924,Y -35.599,Z 157,A -165.6946,B 19.66,C -0.5823,E1 19.5144,E2 253.8202} C_DIS
LIN {X -126.0528,Y -38.7954,Z 157,A -164.2507,B 19.6602,C -0.5779,E1 19.5156,E2 252.3786} C_DIS
LIN {X -124.9898,Y -42.0962,Z 157,A -162.7395,B 19.6602,C -0.5736,E1 19.5169,E2 250.8688} C_DIS
LIN {X -121.939,Y -50.2552,Z 157,A -158.9804,B 19.6606,C -0.5617,E1 19.5206,E2 247.1176} C_DIS
LIN {X -118.7663,Y -57.3514,Z 157,A -155.5288,B 19.6608,C -0.5551,E1 19.5246,E2 243.6613} C_DIS
LIN {X -117.3632,Y -60.1692,Z 157,A -154.1019,B 19.6608,C -0.5536,E1 19.5264,E2 242.2288} C_DIS
LIN {X -115.3494,Y -63.9481,Z 157,A -151.7378,B 19.6605,C -0.5677,E1 19.5297,E2 239.8061} C_DIS
LIN {X -113.1695,Y -67.7314,Z 157,A -150.2542,B 19.661,C -0.5471,E1 19.5317,E2 238.3744} C_DIS
LIN {X -109.2524,Y -73.8833,Z 157,A -147.0871,B 19.6612,C -0.539,E1 19.5365,E2 235.2107} C_DIS
LIN {X -106.7957,Y -77.3918,Z 157,A -145.1933,B 19.6613,C -0.5357,E1 19.5396,E2 233.3147} C_DIS
LIN {X -104.1527,Y -80.9139,Z 157,A -143.2968,B 19.6615,C -0.5305,E1 19.5428,E2 231.4219} C_DIS
LIN {X -101.3485,Y -84.4004,Z 157,A -141.5193,B 19.6617,C -0.5196,E1 19.5459,E2 229.6661} C_DIS
LIN {X -99.152,Y -86.9703,Z 157,A -139.8089,B 19.6616,C -0.5255,E1 19.5491,E2 227.9278} C_DIS
LIN {X -96.201,Y -90.2239,Z 157,A -137.9036,B 19.6616,C -0.5213,E1 19.5527,E2 226.0244} C_DIS
LIN {X -92.9212,Y -93.5969,Z 157,A -135.5999,B 19.6616,C -0.527,E1 19.5573,E2 223.6907} C_DIS
LIN {X -90.3859,Y -96.0481,Z 157,A -134.3718,B 19.6619,C -0.5122,E1 19.5597,E2 222.5005} C_DIS
LIN {X -87.4011,Y -98.7718,Z 157,A -132.5531,B 19.6619,C -0.5112,E1 19.5635,E2 220.6752} C_DIS
LIN {X -84.0749,Y -101.6181,Z 157,A -130.6567,B 19.662,C -0.5074,E1 19.5675,E2 218.7806} C_DIS
LIN {X -80.576,Y -104.4146,Z 157,A -128.6557,B 19.662,C -0.506,E1 19.5719,E2 216.774} C_DIS
LIN {X -76.9515,Y -107.1139,Z 157,A -126.695,B 19.6622,C -0.5026,E1 19.5764,E2 214.8146} C_DIS
LIN {X -73.2957,Y -109.6475,Z 157,A -124.7709,B 19.6622,C -0.4991,E1 19.5808,E2 212.8923} C_DIS
LIN {X -69.7391,Y -111.9432,Z 157,A -122.6274,B 19.662,C -0.5083,E1 19.5859,E2 210.7125} C_DIS
LIN {X -66.5447,Y -113.8715,Z 157,A -121.2789,B 19.6623,C -0.4953,E1 19.5891,E2 209.3977} C_DIS
LIN {X -62.6737,Y -116.0471,Z 157,A -119.3726,B 19.6624,C -0.4918,E1 19.5938,E2 207.4948} C_DIS
LIN {X -59.5971,Y -117.6544,Z 157,A -117.9667,B 19.6626,C -0.4858,E1 19.5972,E2 206.1016} C_DIS
LIN {X -56.5608,Y -119.144,Z 157,A -116.4388,B 19.6626,C -0.4864,E1 19.6011,E2 204.5669} C_DIS
LIN {X -52.7735,Y -120.8698,Z 157,A -114.168,B 19.6622,C -0.5028,E1 19.607,E2 202.2401} C_DIS
LIN {X -48.9008,Y -122.4877,Z 157,A -112.9119,B 19.6627,C -0.4784,E1 19.6101,E2 201.0533} C_DIS
LIN {X -46.2249,Y -123.5216,Z 157,A -111.5546,B 19.6627,C -0.4816,E1 19.6137,E2 199.6825} C_DIS
LIN {X -43.0314,Y -124.6702,Z 157,A -110.0668,B 19.6627,C -0.4809,E1 19.6176,E2 198.1931} C_DIS
LIN {X -37.1631,Y -126.5435,Z 157,A -107.5507,B 19.6629,C -0.4724,E1 19.6243,E2 195.6965} C_DIS
LIN {X -32.0038,Y -127.9466,Z 157,A -105.103,B 19.6628,C -0.476,E1 19.6309,E2 193.2335} C_DIS
LIN {X -28.3622,Y -128.8032,Z 157,A -103.4084,B 19.6628,C -0.4779,E1 19.6355,E2 191.5303} C_DIS
LIN {X -24.7737,Y -129.5402,Z 157,A -101.8773,B 19.6628,C -0.4748,E1 19.6397,E2 190.0062} C_DIS
LIN {X -21.1498,Y -130.1822,Z 157,A -100.038,B 19.6626,C -0.484,E1 19.6449,E2 188.1372} C_DIS
LIN {X -17.1253,Y -130.7713,Z 157,A -98.4979,B 19.6628,C -0.4744,E1 19.6491,E2 186.6242} C_DIS
LIN {X -13.2651,Y -131.2208,Z 157,A -96.6856,B 19.6628,C -0.4792,E1 19.6541,E2 184.7963} C_DIS
LIN {X -9.3601,Y -131.5556,Z 157,A -95.1383,B 19.6628,C -0.4727,E1 19.6584,E2 183.2673} C_DIS
LIN {X -5.7873,Y -131.7626,Z 157,A -93.414,B 19.6628,C -0.4797,E1 19.6632,E2 181.5217} C_DIS
LIN {X -1.6732,Y -131.8785,Z 157,A -91.649,B 19.6628,C -0.479,E1 19.6682,E2 179.7586} C_DIS
LIN {X -1.6732,Y -131.8785,Z 157,A -91.649,B 19.6628,C -0.479,E1 19.6682,E2 179.7586} C_DIS
Enddeposition()
LIN {X 0.9141,Y -130.9507,Z 157,A -90.3735,B 18.345,C -0.3168,E1 18.3499,E2 178.8653} C_DIS
Startdeposition()
$VEL.CP = VEL_PRINT
LIN {X -1.7868,Y -130.945,Z 157,A -92.1501,B 18.3454,C -0.2941,E1 18.3448,E2 180.7139} C_DIS
LIN {X -5.6889,Y -130.8342,Z 157,A -93.9182,B 18.3454,C -0.2918,E1 18.3398,E2 182.4899} C_DIS
LIN {X -9.8256,Y -130.5877,Z 157,A -95.7274,B 18.3454,C -0.292,E1 18.3348,E2 184.2993} C_DIS
LIN {X -13.9681,Y -130.2094,Z 157,A -97.454,B 18.3454,C -0.2957,E1 18.33,E2 186.0154} C_DIS
LIN {X -17.36,Y -129.8011,Z 157,A -98.9431,B 18.3454,C -0.2962,E1 18.3259,E2 187.5044} C_DIS
LIN {X -21.8858,Y -129.115,Z 157,A -100.8895,B 18.3454,C -0.2989,E1 18.3205,E2 189.4445} C_DIS
LIN {X -24.8859,Y -128.5703,Z 157,A -102.3482,B 18.3454,C -0.2949,E1 18.3165,E2 190.9184} C_DIS
LIN {X -29.4499,Y -127.6022,Z 157,A -104.1557,B 18.3452,C -0.3045,E1 18.3116,E2 192.6984} C_DIS
LIN {X -32.1348,Y -126.9523,Z 157,A -105.5229,B 18.3452,C -0.2993,E1 18.3079,E2 194.0847} C_DIS
LIN {X -35.329,Y -126.1007,Z 157,A -106.965,B 18.3452,C -0.3004,E1 18.304,E2 195.5264} C_DIS
LIN {X -40.2627,Y -124.6138,Z 157,A -109.1773,B 18.3452,C -0.3036,E1 18.2981,E2 197.7338} C_DIS
LIN {X -43.3836,Y -123.5622,Z 157,A -110.6628,B 18.3452,C -0.3032,E1 18.2942,E2 199.2246} C_DIS
LIN {X -47.0413,Y -122.2162,Z 157,A -112.5517,B 18.3453,C -0.2981,E1 18.2892,E2 201.1352} C_DIS
LIN {X -52.9653,Y -119.7684,Z 157,A -115.0855,B 18.3451,C -0.3108,E1 18.2827,E2 203.6367} C_DIS
LIN {X -56.8402,Y -117.9782,Z 157,A -117.0774,B 18.3451,C -0.3085,E1 18.2777,E2 205.643} C_DIS
LIN {X -59.8972,Y -116.4564,Z 157,A -118.6491,B 18.3451,C -0.3075,E1 18.2737,E2 207.2237} C_DIS
LIN {X -63.8465,Y -114.3405,Z 157,A -120.671,B 18.3451,C -0.3079,E1 18.2687,E2 209.2524} C_DIS
LIN {X -68.0513,Y -111.8889,Z 157,A -122.9169,B 18.3451,C -0.3069,E1 18.2633,E2 211.5112} C_DIS
LIN {X -70.9815,Y -110.0534,Z 157,A -124.3276,B 18.3451,C -0.3128,E1 18.2601,E2 212.9094} C_DIS
LIN {X -74.724,Y -107.5468,Z 157,A -126.0828,B 18.3449,C -0.3236,E1 18.256,E2 214.6385} C_DIS
LIN {X -77.692,Y -105.4229,Z 157,A -127.8578,B 18.3449,C -0.3199,E1 18.252,E2 216.4338} C_DIS
LIN {X -81.1691,Y -102.77,Z 157,A -129.8092,B 18.3449,C -0.322,E1 18.2477,E2 218.3887} C_DIS
LIN {X -84.5797,Y -99.9818,Z 157,A -131.7511,B 18.3449,C -0.325,E1 18.2435,E2 220.3313} C_DIS
LIN {X -87.7566,Y -97.2053,Z 157,A -133.572,B 18.3448,C -0.3295,E1 18.2397,E2 222.1482} C_DIS
LIN {X -90.8383,Y -94.3319,Z 157,A -135.8308,B 18.345,C -0.3187,E1 18.2351,E2 224.4544} C_DIS
LIN {X -93.7562,Y -91.4325,Z 157,A -136.9943,B 18.3445,C -0.3446,E1 18.2329,E2 225.5421} C_DIS
LIN {X -95.737,Y -89.3556,Z 157,A -138.5187,B 18.3446,C -0.3379,E1 18.2299,E2 227.0972} C_DIS
LIN {X -98.5076,Y -86.2919,Z 157,A -140.3352,B 18.3446,C -0.3416,E1 18.2266,E2 228.9135} C_DIS
LIN {X -101.2562,Y -83.0495,Z 157,A -142.2241,B 18.3446,C -0.3448,E1 18.2232,E2 230.8044} C_DIS
LIN {X -104.0253,Y -79.5532,Z 157,A -144.1673,B 18.3444,C -0.3496,E1 18.2198,E2 232.745} C_DIS
LIN {X -106.7102,Y -75.9146,Z 157,A -146.1726,B 18.3444,C -0.3535,E1 18.2166,E2 234.7517} C_DIS
LIN {X -111.0574,Y -69.3996,Z 157,A -149.4932,B 18.3441,C -0.3657,E1 18.2115,E2 238.0568} C_DIS
LIN {X -114.1913,Y -64.1119,Z 157,A -152.2729,B 18.3441,C -0.3695,E1 18.2076,E2 240.8445} C_DIS
LIN {X -116.0624,Y -60.6551,Z 157,A -153.9788,B 18.344,C -0.3746,E1 18.2053,E2 242.5469} C_DIS
LIN {X -117.619,Y -57.5794,Z 157,A -156.1802,B 18.3443,C -0.3552,E1 18.2025,E2 244.8272} C_DIS
LIN {X -119.8385,Y -52.8085,Z 157,A -157.8687,B 18.3438,C -0.3822,E1 18.2007,E2 246.4421} C_DIS
LIN {X -121.3705,Y -49.1806,Z 157,A -160.4358,B 18.3443,C -0.3587,E1 18.1979,E2 249.1048} C_DIS
LIN {X -123.5708,Y -43.359,Z 157,A -162.1509,B 18.3434,C -0.4003,E1 18.1964,E2 250.7001} C_DIS
LIN {X -124.8331,Y -39.5763,Z 157,A -164.0596,B 18.3434,C -0.3998,E1 18.1947,E2 252.6259} C_DIS
LIN {X -125.9394,Y -35.9057,Z 157,A -165.8477,B 18.3434,C -0.401,E1 18.1933,E2 254.4248} C_DIS
LIN {X -126.9284,Y -32.229,Z 157,A -167.4329,B 18.3433,C -0.4086,E1 18.1922,E2 255.9985} C_DIS
LIN {X -127.8027,Y -28.5725,Z 157,A -169.6167,B 18.3435,C -0.3954,E1 18.1908,E2 258.2427} C_DIS
LIN {X -128.6774,Y -24.326,Z 157,A -170.9496,B 18.343,C -0.4201,E1 18.1901,E2 259.5077} C_DIS
LIN {X -129.1921,Y -21.4235,Z 157,A -172.3441,B 18.343,C -0.4204,E1 18.1894,E2 260.9128} C_DIS
LIN {X -130.1343,Y -14.6656,Z 157,A -175.2327,B 18.3427,C -0.4328,E1 18.1884,E2 263.7861} C_DIS
LIN {X -130.6119,Y -9.4936,Z 157,A -177.6769,B 18.3427,C -0.434,E1 18.1878,E2 266.2471} C_DIS
LIN {X -130.8067,Y -6.27,Z 157,A -179.857,B 18.3432,C -0.4128,E1 18.1875,E2 268.5136} C_DIS
LIN {X -130.9581,Y -0.3052,Z 157,A 177.7377,B 18.3428,C -0.4276,E1 18.1875,E2 270.8918} C_DIS
LIN {X -130.8849,Y 4.3397,Z 157,A 176.3743,B 18.3422,C -0.4563,E1 18.1875,E2 272.1751} C_DIS
LIN {X -130.4638,Y 11.3531,Z 157,A 172.9572,B 18.3422,C -0.4543,E1 18.1882,E2 275.6275} C_DIS
LIN {X -130.0521,Y 15.3639,Z 157,A 171.4035,B 18.3419,C -0.4668,E1 18.1887,E2 277.1542} C_DIS
LIN {X -129.5893,Y 18.876,Z 157,A 169.811,B 18.3419,C -0.4701,E1 18.1893,E2 278.7495} C_DIS
LIN {X -128.5732,Y 24.8712,Z 157,A 167.1165,B 18.3417,C -0.4772,E1 18.1906,E2 281.4438} C_DIS
LIN {X -127.6725,Y 29.1422,Z 157,A 165.2502,B 18.3415,C -0.4845,E1 18.1917,E2 283.3023} C_DIS
Enddeposition()
END
